(* CODESYS project 17.08.01_vi_gwp_library.library
   Title: GWP Library
   Author: ShgB
   Placeholder: GWP Library
   Version: 17.8.1
   Company: Viessmann

Project tree, tasks and I/O mapping:
  libraries: Tc2_Standard, * (Beckhoff Automation GmbH); Tc2_System, * (Beckhoff Automation GmbH); Tc2_Utilities, * (Beckhoff Automation GmbH)
  Allgemein/
    function block Alarm [ST]
    function block COUNT [ST]
    function block MUX_B [ST]
    function block MUX_D_INT [ST]
    function block MUX_D_REAL [ST]
    function block NULL [ST]
    function block SWITCH_INT [ST]
    function block SWITCH_REAL [ST]
    function block Toggle [ST]
  Converters/
    function block Converter2Punkt [ST]
    function block Int_to_Druck [ST]
    function block Int_to_Temperature [ST]
    function block Prozent_to_Int [ST]
    function block Time_to_Timestruct [ST]
    function block Timestruct_to_Time [ST]
  Druck_Temp/
    function block R1234ze [ST]
    function block R134a [ST]
    function block R410a [ST]
  Globale Variablen/
    data type AL_Eintrag
    text list Alarme
    global variables Globale_Uhr
    global variables Nassdampftabelle
    global variables SW_ALZ
    data type SW_Einsatzgrenzen
    global variables Visu
  Handschaltungen/
    function block HS_Bool [ST]
    function block HS_Int [ST]
    function block HS_Real [ST]
  Heizen_Kuehlen/
    function block FG_Heizen [ST]
    function block FG_Kuehlen [ST]
    function block GR_2 [ST]
    function block GR_4_mit_RE [ST]
    function block GR_4_ohne_RE [ST]
    function block REG2_HEIZEN [ST]
    function block REG2_KUEHLEN [ST]
    function block RT_AT_48 [ST]
  Initialisierung/
    function block Globale_Zeit [ST]
  Math/
    function block Average [ST]
    function block Filter [ST]
    function block Maximum [ST]
    function block Minimun [ST]
    function block Range [ST]
    function block Timestruct_Kleiner_Gleich_Timestruct [ST]
  Memory/
    function block Logger [ST]
  Regler/
    function block EEV [ST]
    function block PIDRegler [ST]
    function block PIRegler [ST]
    function block PRegler [ST]
  Timer/
    function block BLINK_A [ST]
    function block BLINK_S [ST]
    function block PULSE [ST]
    function block TOF_Reset [ST]
    function block TON_Reset [ST]
    function block Work [ST]
    function block XPULSE [ST]
  Uhren/
    function block ABS_Bool [ST]
    function block ABS_Int [ST]
    function block ABS_Real [ST]
    function block CLK_D [ST]
    function block CLK_I [ST]
    function block CLK_M [ST]
    function block CLK_W [ST]
    function block CLK_W7 [ST]
    function block CLK_Y [ST]
    function block FerienPRG [ST]
  Verdichter/
    function block Einsatzgrenzen [ST]
    visualisation Einsatzgrenzen
    function block FIFO [ST]
    function block SA_Scroll [ST]
  Version/
    global variables Global_Version
  text list GlobalTextList
*)

// Globale Variablen/AL_Eintrag
TYPE AL_Eintrag :
STRUCT
	x_Aktiv: BOOL;
	i_ID: INT;
	t_TimeOn: DT;
	i_TextIndex: INT;
	t_TimeOff:DT;
END_STRUCT
END_TYPE

// Globale Variablen/SW_Einsatzgrenzen
TYPE SW_Einsatzgrenzen :
STRUCT
	f_SW_EG_MinVerd:REAL;
	f_SW_EG_MaxVerd:REAL;
	f_SW_EG_MinKond:REAL;
	f_SW_EG_MaxKond:REAL;
	f_SW_EG_BVerd:REAL;
	f_SW_EG_BKond:REAL;
	f_SW_EG_CKond:REAL;
	f_SW_EG_DKond:REAL;
	f_SW_EG_EVerd:REAL;
	f_SW_EG_FVerd:REAL;
	f_SW_EG_GKond:REAL;
END_STRUCT
END_TYPE

// Globale Variablen/Globale_Uhr
{attribute 'qualified_only'}
VAR_GLOBAL
//aktuelle Uhrzeit
	   systemtimestruct	:timestruct;   
	   systemDateAndTime:dt;
END_VAR

// Globale Variablen/Nassdampftabelle
{attribute 'qualified_only'}
VAR_GLOBAL
END_VAR
VAR_GLOBAL CONSTANT
	// Arrayposition entspricht dem absoluten Druck. Z.B. 1.00bara => 0.00bar Überdruck => Arrayposition 100
	R410a: ARRAY [0..5100] OF INT := [-805,-802,-799,-796,-799,-795,-792,-789,-785,-782,-779,-776,-772,-769,-766,-762,-759,-756,-752,-749,-746,-743,-739,-736,-733,-729,-726,-723,-719,-716,-713,-710,-706,-703,-700,-703,-698,-694,-690,-685,-681,-677,-673,-669,-666,-662,-658,-654,-651,-647,-644,-641,-637,-634,-631,-628,-624,-621,-618,-615,-612,-609,-606,-604,-601,-598,-595,-592,-590,-587,-585,-582,-579,-577,-574,-572,-569,-567,-565,-562,-560,-558,-555,-553,-551,-548,-546,-544,-542,-540,-537,-535,-533,-531,-529,-527,-525,-523,-521,-519,-517,-515,-513,-511,-509,-507,-506,-504,-502,-500,-498,-496,-495,-493,-491,-489,-488,-486,-484,-482,-481,-479,-477,-476,-474,-472,-471,-469,-467,-466,-464,-463,-461,-459,-458,-456,-455,-453,-452,-450,-449,-447,-446,-444,-443,-441,-440,-438,-437,-436,-434,-433,-431,-430,-428,-427,-426,-424,-423,-422,-420,-419,-418,-416,-415,-414,-412,-411,-410,-408,-407,-406,-404,-403,-402,-401,-399,-398,-397,-396,-394,-393,-392,-391,-390,-388,-387,-386,-385,-384,-382,-381,-380,-379,-378,-377,-375,-374,-373,-372,-371,-370,-369,-367,-366,-365,-364,-363,-362,-361,-360,-359,-357,-356,-355,-354,-353,-352,-351,-350,-349,-348,-347,-346,-345,-344,-343,-342,-341,-340,-339,-338,-337,-336,-335,-334,-333,-332,-331,-330,-329,-328,-327,-326,-325,-324,-323,-322,-321,-320,-319,-318,-317,-316,-315,-314,-313,-312,-311,-310,-309,-309,-308,-307,-306,-305,-304,-303,-302,-301,-300,-299,-299,-298,-297,-296,-295,-294,-293,-292,-291,-291,-290,-289,-288,-287,-286,-285,-285,-284,-283,-282,-281,-280,-279,-279,-278,-277,-276,-275,-274,-274,-273,-272,-271,-270,-269,-269,-268,-267,-266,-265,-265,-264,-263,-262,-261,-261,-260,-259,-258,-257,-257,-256,-255,-254,-254,-253,-252,-251,-250,-250,-249,-248,-247,-247,-246,-245,-244,-244,-243,-242,-241,-241,-240,-239,-238,-238,-237,-236,-235,-235,-234,-233,-232,-232,-231,-230,-230,-229,-228,-227,-227,-226,-225,-225,-224,-223,-222,-222,-221,-220,-220,-219,-218,-218,-217,-216,-215,-215,-214,-213,-213,-212,-211,-211,-210,-209,-209,-208,-207,-207,-206,-205,-204,-204,-203,-202,-202,-201,-200,-200,-199,-199,-198,-197,-197,-196,-195,-195,-194,-193,-193,-192,-191,-191,-190,-189,-189,-188,-187,-187,-186,-186,-185,-184,-184,-183,-182,-182,-181,-180,-180,-179,-179,-178,-177,-177,-176,-176,-175,-174,-174,-173,-172,-172,-171,-171,-170,-169,-169,-168,-168,-167,-166,-166,-165,-165,-164,-163,-163,-162,-162,-161,-160,-160,-159,-159,-158,-157,-157,-156,-156,-155,-154,-154,-153,-153,-152,-152,-151,-150,-150,-149,-149,-148,-148,-147,-146,-146,-145,-145,-144,-144,-143,-142,-142,-141,-141,-140,-140,-139,-139,-138,-137,-137,-136,-136,-135,-135,-134,-134,-133,-132,-132,-131,-131,-130,-130,-129,-129,-128,-128,-127,-126,-126,-125,-125,-124,-124,-123,-123,-122,-122,-121,-121,-120,-119,-119,-118,-118,-117,-117,-116,-116,-115,-115,-114,-114,-113,-113,-112,-112,-111,-111,-110,-110,-109,-108,-108,-107,-107,-106,-106,-105,-105,-104,-104,-103,-103,-102,-102,-101,-101,-100,-100,-99,-99,-98,-98,-97,-97,-96,-96,-95,-95,-94,-94,-93,-93,-92,-92,-91,-91,-90,-90,-89,-89,-88,-88,-87,-87,-86,-86,-86,-85,-85,-84,-84,-83,-83,-82,-82,-81,-81,-80,-80,-79,-79,-78,-78,-77,-77,-76,-76,-75,-75,-75,-74,-74,-73,-73,-72,-72,-71,-71,-70,-70,-69,-69,-68,-68,-68,-67,-67,-66,-66,-65,-65,-64,-64,-63,-63,-62,-62,-62,-61,-61,-60,-60,-59,-59,-58,-58,-57,-57,-57,-56,-56,-55,-55,-54,-54,-53,-53,-53,-52,-52,-51,-51,-50,-50,-49,-49,-49,-48,-48,-47,-47,-46,-46,-45,-45,-45,-44,-44,-43,-43,-42,-42,-42,-41,-41,-40,-40,-39,-39,-39,-38,-38,-37,-37,-36,-36,-35,-35,-35,-34,-34,-33,-33,-33,-32,-32,-31,-31,-30,-30,-30,-29,-29,-28,-28,-27,-27,-27,-26,-26,-25,-25,-25,-24,-24,-23,-23,-22,-22,-22,-21,-21,-20,-20,-20,-19,-19,-18,-18,-18,-17,-17,-16,-16,-15,-15,-15,-14,-14,-13,-13,-13,-12,-12,-11,-11,-11,-10,-10,-9,-9,-9,-8,-8,-7,-7,-7,-6,-6,-5,-5,-5,-4,-4,-3,-3,-3,-2,-2,-2,-1,-1,0,0,1,1,1,2,2,3,3,3,4,4,4,5,5,6,6,6,7,7,8,8,8,9,9,9,10,10,11,11,11,12,12,13,13,13,14,14,14,15,15,16,16,16,17,17,17,18,18,19,19,19,20,20,20,21,21,22,22,22,23,23,23,24,24,25,25,25,26,26,26,27,27,27,28,28,29,29,29,30,30,30,31,31,31,32,32,33,33,33,34,34,34,35,35,35,36,36,37,37,37,38,38,38,39,39,39,40,40,40,41,41,42,42,42,43,43,43,44,44,44,45,45,45,46,46,46,47,47,48,48,48,49,49,49,50,50,50,51,51,51,52,52,52,53,53,53,54,54,54,55,55,56,56,56,57,57,57,58,58,58,59,59,59,60,60,60,61,61,61,62,62,62,63,63,63,64,64,64,65,65,65,66,66,66,67,67,67,68,68,68,69,69,69,70,70,70,71,71,71,72,72,72,73,73,73,74,74,74,75,75,75,76,76,76,77,77,77,78,78,78,79,79,79,80,80,80,81,81,81,82,82,82,83,83,83,83,84,84,84,85,85,85,86,86,86,87,87,87,88,88,88,89,89,89,90,90,90,91,91,91,91,92,92,92,93,93,93,94,94,94,95,95,95,96,96,96,97,97,97,97,98,98,98,99,99,99,100,100,100,101,101,101,101,102,102,102,103,103,103,104,104,104,105,105,105,105,106,106,106,107,107,107,108,108,108,109,109,109,109,110,110,110,111,111,111,112,112,112,113,113,113,113,114,114,114,115,115,115,116,116,116,116,117,117,117,118,118,118,119,119,119,119,120,120,120,121,121,121,121,122,122,122,123,123,123,124,124,124,124,125,125,125,126,126,126,127,127,127,127,128,128,128,129,129,129,129,130,130,130,131,131,131,131,132,132,132,133,133,133,133,134,134,134,135,135,135,136,136,136,136,137,137,137,138,138,138,138,139,139,139,140,140,140,140,141,141,141,142,142,142,142,143,143,143,143,144,144,144,145,145,145,145,146,146,146,147,147,147,147,148,148,148,149,149,149,149,150,150,150,151,151,151,151,152,152,152,152,153,153,153,154,154,154,154,155,155,155,155,156,156,156,157,157,157,157,158,158,158,159,159,159,159,160,160,160,160,161,161,161,162,162,162,162,163,163,163,163,164,164,164,164,165,165,165,166,166,166,166,167,167,167,167,168,168,168,169,169,169,169,170,170,170,170,171,171,171,171,172,172,172,173,173,173,173,174,174,174,174,175,175,175,175,176,176,176,177,177,177,177,178,178,178,178,179,179,179,179,180,180,180,180,181,181,181,181,182,182,182,183,183,183,183,184,184,184,184,185,185,185,185,186,186,186,186,187,187,187,187,188,188,188,188,189,189,189,189,190,190,190,191,191,191,191,192,192,192,192,193,193,193,193,194,194,194,194,195,195,195,195,196,196,196,196,197,197,197,197,198,198,198,198,199,199,199,199,200,200,200,200,201,201,201,201,202,202,202,202,203,203,203,203,204,204,204,204,205,205,205,205,206,206,206,206,207,207,207,207,208,208,208,208,209,209,209,209,210,210,210,210,211,211,211,211,212,212,212,212,213,213,213,213,214,214,214,214,214,215,215,215,215,216,216,216,216,217,217,217,217,218,218,218,218,219,219,219,219,220,220,220,220,221,221,221,221,221,222,222,222,222,223,223,223,223,224,224,224,224,225,225,225,225,226,226,226,226,227,227,227,227,227,228,228,228,228,229,229,229,229,230,230,230,230,231,231,231,231,231,232,232,232,232,233,233,233,233,234,234,234,234,235,235,235,235,235,236,236,236,236,237,237,237,237,238,238,238,238,238,239,239,239,239,240,240,240,240,241,241,241,241,241,242,242,242,242,243,243,243,243,244,244,244,244,244,245,245,245,245,246,246,246,246,247,247,247,247,247,248,248,248,248,249,249,249,249,249,250,250,250,250,251,251,251,251,252,252,252,252,252,253,253,253,253,254,254,254,254,254,255,255,255,255,256,256,256,256,256,257,257,257,257,258,258,258,258,258,259,259,259,259,260,260,260,260,260,261,261,261,261,262,262,262,262,262,263,263,263,263,264,264,264,264,264,265,265,265,265,266,266,266,266,266,267,267,267,267,268,268,268,268,268,269,269,269,269,270,270,270,270,270,271,271,271,271,271,272,272,272,272,273,273,273,273,273,274,274,274,274,275,275,275,275,275,276,276,276,276,276,277,277,277,277,278,278,278,278,278,279,279,279,279,279,280,280,280,280,281,281,281,281,281,282,282,282,282,282,283,283,283,283,283,284,284,284,284,285,285,285,285,285,286,286,286,286,286,287,287,287,287,288,288,288,288,288,289,289,289,289,289,290,290,290,290,290,291,291,291,291,291,292,292,292,292,293,293,293,293,293,294,294,294,294,294,295,295,295,295,295,296,296,296,296,296,297,297,297,297,298,298,298,298,298,299,299,299,299,299,300,300,300,300,300,301,301,301,301,301,302,302,302,302,302,303,303,303,303,303,304,304,304,304,304,305,305,305,305,305,306,306,306,306,307,307,307,307,307,308,308,308,308,308,309,309,309,309,309,310,310,310,310,310,311,311,311,311,311,312,312,312,312,312,313,313,313,313,313,314,314,314,314,314,315,315,315,315,315,316,316,316,316,316,317,317,317,317,317,318,318,318,318,318,319,319,319,319,319,320,320,320,320,320,321,321,321,321,321,322,322,322,322,322,322,323,323,323,323,323,324,324,324,324,324,325,325,325,325,325,326,326,326,326,326,327,327,327,327,327,328,328,328,328,328,329,329,329,329,329,330,330,330,330,330,330,331,331,331,331,331,332,332,332,332,332,333,333,333,333,333,334,334,334,334,334,335,335,335,335,335,336,336,336,336,336,336,337,337,337,337,337,338,338,338,338,338,339,339,339,339,339,340,340,340,340,340,340,341,341,341,341,341,342,342,342,342,342,343,343,343,343,343,344,344,344,344,344,344,345,345,345,345,345,346,346,346,346,346,347,347,347,347,347,347,348,348,348,348,348,349,349,349,349,349,350,350,350,350,350,350,351,351,351,351,351,352,352,352,352,352,352,353,353,353,353,353,354,354,354,354,354,355,355,355,355,355,355,356,356,356,356,356,357,357,357,357,357,357,358,358,358,358,358,359,359,359,359,359,360,360,360,360,360,360,361,361,361,361,361,362,362,362,362,362,362,363,363,363,363,363,364,364,364,364,364,364,365,365,365,365,365,366,366,366,366,366,366,367,367,367,367,367,368,368,368,368,368,368,369,369,369,369,369,370,370,370,370,370,370,371,371,371,371,371,371,372,372,372,372,372,373,373,373,373,373,373,374,374,374,374,374,375,375,375,375,375,375,376,376,376,376,376,376,377,377,377,377,377,378,378,378,378,378,378,379,379,379,379,379,379,380,380,380,380,380,381,381,381,381,381,381,382,382,382,382,382,382,383,383,383,383,383,384,384,384,384,384,384,385,385,385,385,385,385,386,386,386,386,386,387,387,387,387,387,387,388,388,388,388,388,388,389,389,389,389,389,389,390,390,390,390,390,391,391,391,391,391,391,392,392,392,392,392,392,393,393,393,393,393,393,394,394,394,394,394,394,395,395,395,395,395,395,396,396,396,396,396,397,397,397,397,397,397,398,398,398,398,398,398,399,399,399,399,399,399,400,400,400,400,400,400,401,401,401,401,401,401,402,402,402,402,402,402,403,403,403,403,403,404,404,404,404,404,404,405,405,405,405,405,405,406,406,406,406,406,406,407,407,407,407,407,407,408,408,408,408,408,408,409,409,409,409,409,409,410,410,410,410,410,410,411,411,411,411,411,411,412,412,412,412,412,412,413,413,413,413,413,413,414,414,414,414,414,414,415,415,415,415,415,415,416,416,416,416,416,416,417,417,417,417,417,417,418,418,418,418,418,418,418,419,419,419,419,419,419,420,420,420,420,420,420,421,421,421,421,421,421,422,422,422,422,422,422,423,423,423,423,423,423,424,424,424,424,424,424,425,425,425,425,425,425,426,426,426,426,426,426,426,427,427,427,427,427,427,428,428,428,428,428,428,429,429,429,429,429,429,430,430,430,430,430,430,431,431,431,431,431,431,431,432,432,432,432,432,432,433,433,433,433,433,433,434,434,434,434,434,434,435,435,435,435,435,435,435,436,436,436,436,436,436,437,437,437,437,437,437,438,438,438,438,438,438,439,439,439,439,439,439,439,440,440,440,440,440,440,441,441,441,441,441,441,442,442,442,442,442,442,442,443,443,443,443,443,443,444,444,444,444,444,444,445,445,445,445,445,445,445,446,446,446,446,446,446,447,447,447,447,447,447,447,448,448,448,448,448,448,449,449,449,449,449,449,450,450,450,450,450,450,450,451,451,451,451,451,451,452,452,452,452,452,452,452,453,453,453,453,453,453,454,454,454,454,454,454,454,455,455,455,455,455,455,456,456,456,456,456,456,456,457,457,457,457,457,457,458,458,458,458,458,458,458,459,459,459,459,459,459,460,460,460,460,460,460,460,461,461,461,461,461,461,461,462,462,462,462,462,462,463,463,463,463,463,463,463,464,464,464,464,464,464,465,465,465,465,465,465,465,466,466,466,466,466,466,466,467,467,467,467,467,467,468,468,468,468,468,468,468,469,469,469,469,469,469,469,470,470,470,470,470,470,471,471,471,471,471,471,471,472,472,472,472,472,472,472,473,473,473,473,473,473,474,474,474,474,474,474,474,475,475,475,475,475,475,475,476,476,476,476,476,476,476,477,477,477,477,477,477,478,478,478,478,478,478,478,479,479,479,479,479,479,479,480,480,480,480,480,480,480,481,481,481,481,481,481,482,482,482,482,482,482,482,483,483,483,483,483,483,483,484,484,484,484,484,484,484,485,485,485,485,485,485,485,486,486,486,486,486,486,486,487,487,487,487,487,487,487,488,488,488,488,488,488,488,489,489,489,489,489,489,490,490,490,490,490,490,490,491,491,491,491,491,491,491,492,492,492,492,492,492,492,493,493,493,493,493,493,493,494,494,494,494,494,494,494,495,495,495,495,495,495,495,496,496,496,496,496,496,496,497,497,497,497,497,497,497,498,498,498,498,498,498,498,499,499,499,499,499,499,499,500,500,500,500,500,500,500,501,501,501,501,501,501,501,502,502,502,502,502,502,502,503,503,503,503,503,503,503,504,504,504,504,504,504,504,504,505,505,505,505,505,505,505,506,506,506,506,506,506,506,507,507,507,507,507,507,507,508,508,508,508,508,508,508,509,509,509,509,509,509,509,510,510,510,510,510,510,510,511,511,511,511,511,511,511,511,512,512,512,512,512,512,512,513,513,513,513,513,513,513,514,514,514,514,514,514,514,515,515,515,515,515,515,515,516,516,516,516,516,516,516,516,517,517,517,517,517,517,517,518,518,518,518,518,518,518,519,519,519,519,519,519,519,519,520,520,520,520,520,520,520,521,521,521,521,521,521,521,522,522,522,522,522,522,522,523,523,523,523,523,523,523,523,524,524,524,524,524,524,524,525,525,525,525,525,525,525,525,526,526,526,526,526,526,526,527,527,527,527,527,527,527,528,528,528,528,528,528,528,528,529,529,529,529,529,529,529,530,530,530,530,530,530,530,530,531,531,531,531,531,531,531,532,532,532,532,532,532,532,533,533,533,533,533,533,533,533,534,534,534,534,534,534,534,535,535,535,535,535,535,535,535,536,536,536,536,536,536,536,537,537,537,537,537,537,537,537,538,538,538,538,538,538,538,538,539,539,539,539,539,539,539,540,540,540,540,540,540,540,540,541,541,541,541,541,541,541,542,542,542,542,542,542,542,542,543,543,543,543,543,543,543,544,544,544,544,544,544,544,544,545,545,545,545,545,545,545,545,546,546,546,546,546,546,546,547,547,547,547,547,547,547,547,548,548,548,548,548,548,548,548,549,549,549,549,549,549,549,550,550,550,550,550,550,550,550,551,551,551,551,551,551,551,551,552,552,552,552,552,552,552,553,553,553,553,553,553,553,553,554,554,554,554,554,554,554,554,555,555,555,555,555,555,555,555,556,556,556,556,556,556,556,556,557,557,557,557,557,557,557,558,558,558,558,558,558,558,558,559,559,559,559,559,559,559,559,560,560,560,560,560,560,560,560,561,561,561,561,561,561,561,561,562,562,562,562,562,562,562,562,563,563,563,563,563,563,563,564,564,564,564,564,564,564,564,565,565,565,565,565,565,565,565,566,566,566,566,566,566,566,566,567,567,567,567,567,567,567,567,568,568,568,568,568,568,568,568,569,569,569,569,569,569,569,569,570,570,570,570,570,570,570,570,571,571,571,571,571,571,571,571,572,572,572,572,572,572,572,572,573,573,573,573,573,573,573,573,574,574,574,574,574,574,574,574,575,575,575,575,575,575,575,575,576,576,576,576,576,576,576,576,577,577,577,577,577,577,577,577,578,578,578,578,578,578,578,578,579,579,579,579,579,579,579,579,580,580,580,580,580,580,580,580,580,581,581,581,581,581,581,581,581,582,582,582,582,582,582,582,582,583,583,583,583,583,583,583,583,584,584,584,584,584,584,584,584,585,585,585,585,585,585,585,585,586,586,586,586,586,586,586,586,586,587,587,587,587,587,587,587,587,588,588,588,588,588,588,588,588,589,589,589,589,589,589,589,589,590,590,590,590,590,590,590,590,590,591,591,591,591,591,591,591,591,592,592,592,592,592,592,592,592,593,593,593,593,593,593,593,593,593,594,594,594,594,594,594,594,594,595,595,595,595,595,595,595,595,596,596,596,596,596,596,596,596,596,597,597,597,597,597,597,597,597,598,598,598,598,598,598,598,598,599,599,599,599,599,599,599,599,599,600,600,600,600,600,600,600,600,601,601,601,601,601,601,601,601,601,602,602,602,602,602,602,602,602,603,603,603,603,603,603,603,603,604,604,604,604,604,604,604,604,604,605,605,605,605,605,605,605,605,606,606,606,606,606,606,606,606,606,607,607,607,607,607,607,607,607,608,608,608,608,608,608,608,608,608,609,609,609,609,609,609,609,609,609,610,610,610,610,610,610,610,610,611,611,611,611,611,611,611,611,611,612,612,612,612,612,612,612,612,613,613,613,613,613,613,613,613,613,614,614,614,614,614,614,614,614,614,615,615,615,615,615,615,615,615,616,616,616,616,616,616,616,616,616,617,617,617,617,617,617,617,617,617,618,618,618,618,618,618,618,618,619,619,619,619,619,619,619,619,619,620,620,620,620,620,620,620,620,620,621,621,621,621,621,621,621,621,622,622,622,622,622,622,622,622,622,623,623,623,623,623,623,623,623,623,624,624,624,624,624,624,624,624,624,625,625,625,625,625,625,625,625,625,626,626,626,626,626,626,626,626,627,627,627,627,627,627,627,627,627,628,628,628,628,628,628,628,628,628,629,629,629,629,629,629,629,629,629,630,630,630,630,630,630,630,630,630,631,631,631,631,631,631,631,631,631,632,632,632,632,632,632,632,632,632,633,633,633,633,633,633,633,633,633,634,634,634,634,634,634,634,634,634,635,635,635,635,635,635,635,635,635,636,636,636,636,636,636,636,636,636,637,637,637,637,637,637,637,637,637,638,638,638,638,638,638,638,638,638,639,639,639,639,639,639,639,639,639,640,640,640,640,640,640,640,640,640,641,641,641,641,641,641,641,641,641,642,642,642,642,642,642,642,642,642,643,643,643,643,643,643,643,643,643,644,644,644,644,644,644,644,644,644,645,645,645,645,645,645,645,645,645,646,646,646,646,646,646,646,646,646,647,647,647,647,647,647,647,647,647,648,648,648,648,648,648,648,648,648,648,649,649,649,649,649,649,649,649,649,650,650,650,650,650,650,650,650,650,651,651,651,651,651,651,651,651,651,652,652,652,652,652,652,652,652,652,652,653,653,653,653,653,653,653,653,653,654,654,654,654,654,654,654,654,654,655,655,655,655,655,655,655,655,655,656,656,656,656,656,656,656,656,656,656,657,657,657,657,657,657,657,657,657,658,658,658,658,658,658,658,658,658,659,659,659,659,659,659,659,659,659,659,660,660,660,660,660,660,660,660,660,661,661,661,661,661,661,661,661,661,661,662,662,662,662,662,662,662,662,662,663,663,663,663,663,663,663,663,663,664,664,664,664,664,664,664,664,664,664,665,665,665,665,665,665,665,665,665,666,666,666,666,666,666,666,666,666,666,667,667,667,667,667,667,667,667,667,668,668,668,668,668,668,668,668,668,668,669,669,669,669,669,669,669,669,669,670,670,670,670,670,670,670,670,670,670,671,671,671,671,671,671,671,671,671,671,672,672,672,672,672,672,672,672,672,673,673,673,673,673,673,673,673,673,673,674,674,674,674,674,674,674,674,674,675,675,675,675,675,675,675,675,675,675,676,676,676,676,676,676,676,676,676,676,677,677,677,677,677,677,677,677,677,678,678,678,678,678,678,678,678,678,678,679,679,679,679,679,679,679,679,679,679,680,680,680,680,680,680,680,680,680,680,681,681,681,681,681,681,681,681,681,682,682,682,682,682,682,682,682,682,682,683,683,683,683,683,683,683,683,683,683,684,684,684,684,684,684,684,684,684,684,685,685,685,685,685,685,685,685,685,685,686,686,686,686,686,686,686,686,686,686,687,687,687,687,687,687,687,687,687,688,688,688,688,688,688,688,688,688,688,689,689,689,689,689,689,689,689,689,689,690,690,690,690,690,690,690,690,690,690,691,691,691,691,691,691,691,691,691,691,692,692,692,692,692,692,692,692,692,692,693,693,693,693,693,693,693,693,693,693,694,694,694,694,694,694,694,694,694,694,695,695,695,695,695,695,695,695,695,695,696,696,696,696,696,696,696,696,696,696,697,697,697,697,697,697,697,697,697,697,698,698,698,698,698,698,698,698,698,698,699,699,699,699,699,699,699,699,699,699,700,700,700,700,700,700,700,700,700,700,701,701,701,701,701,701,701,701,701,701,702,702,702,702,702,702,702,702,702,702,703,703,703,703,703,703,703,703,703,703,704,704,704,704,704,704,704,704,704,704,705,705,705,705,705,705,705,705,705,705,706,706,706,706,706,706,706,706,706,706,707,707,707,707,707,707,707,707,707,707,708,708,708,708,708,708,708,708,708,708,709,709,709,709,709,709,709,709,709,709,710,710,710,710,710,710,710,710,710,710,711,711,711,711,711,711,711,711,711,711,712,712,712,712,712,712,712,712,712,712,713,713,713,713,713,713,713,713,713,713,714];
	// Arrayposition entspricht dem absoluten Druck. Z.B. 1.00bara => 0.00bar Überdruck => Arrayposition 100
	R1234ze: ARRAY [0..5100] OF INT := [-483,-481,-478,-475,-472,-470,-467,-464,-461,-459,-456,-453,-450,-448,-445,-442,-439,-437,-434,-431,-428,-426,-423,-420,-477,-470,-463,-456,-450,-443,-437,-431,-426,-420,-414,-409,-404,-399,-394,-389,-384,-379,-375,-370,-366,-361,-357,-353,-349,-345,-341,-337,-333,-329,-325,-322,-318,-314,-311,-307,-304,-300,-297,-294,-290,-287,-284,-281,-278,-275,-272,-268,-266,-263,-260,-257,-254,-251,-248,-245,-243,-240,-237,-235,-232,-229,-227,-224,-222,-219,-217,-214,-212,-209,-207,-204,-202,-200,-197,-195,-193,-191,-188,-186,-184,-182,-179,-177,-175,-173,-171,-169,-167,-164,-162,-160,-158,-156,-154,-152,-150,-148,-146,-144,-142,-140,-139,-137,-135,-133,-131,-129,-127,-125,-124,-122,-120,-118,-116,-115,-113,-111,-109,-108,-106,-104,-102,-101,-99,-97,-96,-94,-92,-91,-89,-88,-86,-84,-83,-81,-79,-78,-76,-75,-73,-72,-70,-69,-67,-66,-64,-62,-61,-59,-58,-57,-55,-54,-52,-51,-49,-48,-46,-45,-43,-42,-41,-39,-38,-36,-35,-34,-32,-31,-30,-28,-27,-25,-24,-23,-21,-20,-19,-17,-16,-15,-14,-12,-11,-10,-8,-7,-6,-5,-3,-2,-1,1,2,3,4,6,7,8,9,10,12,13,14,15,17,18,19,20,21,22,24,25,26,27,28,29,31,32,33,34,35,36,37,39,40,41,42,43,44,45,46,47,49,50,51,52,53,54,55,56,57,58,59,60,62,63,64,65,66,67,68,69,70,71,72,73,74,75,76,77,78,79,80,81,82,83,84,85,86,87,88,89,90,91,92,93,94,95,96,97,98,99,100,101,102,103,104,104,105,106,107,108,109,110,111,112,113,114,115,116,117,117,118,119,120,121,122,123,124,125,126,127,127,128,129,130,131,132,133,134,134,135,136,137,138,139,140,141,141,142,143,144,145,146,147,147,148,149,150,151,152,152,153,154,155,156,157,157,158,159,160,161,162,162,163,164,165,166,166,167,168,169,170,170,171,172,173,174,174,175,176,177,178,178,179,180,181,181,182,183,184,185,185,186,187,188,188,189,190,191,192,192,193,194,195,195,196,197,198,198,199,200,201,201,202,203,204,204,205,206,206,207,208,209,209,210,211,212,212,213,214,214,215,216,217,217,218,219,219,220,221,222,222,223,224,224,225,226,227,227,228,229,229,230,231,231,232,233,233,234,235,236,236,237,238,238,239,240,240,241,242,242,243,244,244,245,246,246,247,248,248,249,250,250,251,252,252,253,254,254,255,256,256,257,258,258,259,260,260,261,261,262,263,263,264,265,265,266,267,267,268,269,269,270,270,271,272,272,273,274,274,275,275,276,277,277,278,279,279,280,280,281,282,282,283,284,284,285,285,286,287,287,288,288,289,290,290,291,291,292,293,293,294,294,295,296,296,297,297,298,299,299,300,300,301,302,302,303,303,304,305,305,306,306,307,308,308,309,309,310,310,311,312,312,313,313,314,314,315,316,316,317,317,318,318,319,320,320,321,321,322,322,323,324,324,325,325,326,326,327,327,328,329,329,330,330,331,331,332,332,333,334,334,335,335,336,336,337,337,338,339,339,340,340,341,341,342,342,343,343,344,344,345,346,346,347,347,348,348,349,349,350,350,351,351,352,352,353,354,354,355,355,356,356,357,357,358,358,359,359,360,360,361,361,362,362,363,363,364,365,365,366,366,367,367,368,368,369,369,370,370,371,371,372,372,373,373,374,374,375,375,376,376,377,377,378,378,379,379,380,380,381,381,382,382,383,383,384,384,385,385,386,386,387,387,388,388,389,389,390,390,391,391,392,392,393,393,394,394,395,395,395,396,396,397,397,398,398,399,399,400,400,401,401,402,402,403,403,404,404,405,405,406,406,407,407,407,408,408,409,409,410,410,411,411,412,412,413,413,414,414,414,415,415,416,416,417,417,418,418,419,419,420,420,421,421,421,422,422,423,423,424,424,425,425,426,426,426,427,427,428,428,429,429,430,430,431,431,431,432,432,433,433,434,434,435,435,435,436,436,437,437,438,438,439,439,439,440,440,441,441,442,442,443,443,443,444,444,445,445,446,446,447,447,447,448,448,449,449,450,450,450,451,451,452,452,453,453,453,454,454,455,455,456,456,456,457,457,458,458,459,459,459,460,460,461,461,462,462,462,463,463,464,464,465,465,465,466,466,467,467,467,468,468,469,469,470,470,470,471,471,472,472,472,473,473,474,474,475,475,475,476,476,477,477,477,478,478,479,479,479,480,480,481,481,482,482,482,483,483,484,484,484,485,485,486,486,486,487,487,488,488,488,489,489,490,490,490,491,491,492,492,492,493,493,494,494,494,495,495,496,496,496,497,497,498,498,498,499,499,500,500,500,501,501,502,502,502,503,503,503,504,504,505,505,505,506,506,507,507,507,508,508,509,509,509,510,510,510,511,511,512,512,512,513,513,514,514,514,515,515,515,516,516,517,517,517,518,518,519,519,519,520,520,520,521,521,522,522,522,523,523,523,524,524,525,525,525,526,526,526,527,527,528,528,528,529,529,529,530,530,531,531,531,532,532,532,533,533,534,534,534,535,535,535,536,536,536,537,537,538,538,538,539,539,539,540,540,540,541,541,542,542,542,543,543,543,544,544,544,545,545,546,546,546,547,547,547,548,548,548,549,549,550,550,550,551,551,551,552,552,552,553,553,553,554,554,555,555,555,556,556,556,557,557,557,558,558,558,559,559,559,560,560,561,561,561,562,562,562,563,563,563,564,564,564,565,565,565,566,566,566,567,567,568,568,568,569,569,569,570,570,570,571,571,571,572,572,572,573,573,573,574,574,574,575,575,575,576,576,576,577,577,577,578,578,579,579,579,580,580,580,581,581,581,582,582,582,583,583,583,584,584,584,585,585,585,586,586,586,587,587,587,588,588,588,589,589,589,590,590,590,591,591,591,592,592,592,593,593,593,594,594,594,595,595,595,596,596,596,597,597,597,598,598,598,599,599,599,600,600,600,601,601,601,601,602,602,602,603,603,603,604,604,604,605,605,605,606,606,606,607,607,607,608,608,608,609,609,609,610,610,610,611,611,611,612,612,612,612,613,613,613,614,614,614,615,615,615,616,616,616,617,617,617,618,618,618,619,619,619,619,620,620,620,621,621,621,622,622,622,623,623,623,624,624,624,625,625,625,625,626,626,626,627,627,627,628,628,628,629,629,629,629,630,630,630,631,631,631,632,632,632,633,633,633,634,634,634,634,635,635,635,636,636,636,637,637,637,638,638,638,638,639,639,639,640,640,640,641,641,641,641,642,642,642,643,643,643,644,644,644,644,645,645,645,646,646,646,647,647,647,648,648,648,648,649,649,649,650,650,650,651,651,651,651,652,652,652,653,653,653,653,654,654,654,655,655,655,656,656,656,656,657,657,657,658,658,658,659,659,659,659,660,660,660,661,661,661,661,662,662,662,663,663,663,664,664,664,664,665,665,665,666,666,666,666,667,667,667,668,668,668,668,669,669,669,670,670,670,670,671,671,671,672,672,672,673,673,673,673,674,674,674,675,675,675,675,676,676,676,677,677,677,677,678,678,678,679,679,679,679,680,680,680,681,681,681,681,682,682,682,683,683,683,683,684,684,684,684,685,685,685,686,686,686,686,687,687,687,688,688,688,688,689,689,689,690,690,690,690,691,691,691,691,692,692,692,693,693,693,693,694,694,694,695,695,695,695,696,696,696,696,697,697,697,698,698,698,698,699,699,699,700,700,700,700,701,701,701,701,702,702,702,703,703,703,703,704,704,704,704,705,705,705,706,706,706,706,707,707,707,707,708,708,708,709,709,709,709,710,710,710,710,711,711,711,711,712,712,712,713,713,713,713,714,714,714,714,715,715,715,716,716,716,716,717,717,717,717,718,718,718,718,719,719,719,719,720,720,720,721,721,721,721,722,722,722,722,723,723,723,723,724,724,724,725,725,725,725,726,726,726,726,727,727,727,727,728,728,728,728,729,729,729,730,730,730,730,731,731,731,731,732,732,732,732,733,733,733,733,734,734,734,734,735,735,735,735,736,736,736,737,737,737,737,738,738,738,738,739,739,739,739,740,740,740,740,741,741,741,741,742,742,742,742,743,743,743,743,744,744,744,744,745,745,745,745,746,746,746,746,747,747,747,748,748,748,748,749,749,749,749,750,750,750,750,751,751,751,751,752,752,752,752,753,753,753,753,754,754,754,754,755,755,755,755,756,756,756,756,757,757,757,757,758,758,758,758,759,759,759,759,760,760,760,760,761,761,761,761,762,762,762,762,763,763,763,763,764,764,764,764,764,765,765,765,765,766,766,766,766,767,767,767,767,768,768,768,768,769,769,769,769,770,770,770,770,771,771,771,771,772,772,772,772,773,773,773,773,774,774,774,774,775,775,775,775,775,776,776,776,776,777,777,777,777,778,778,778,778,779,779,779,779,780,780,780,780,781,781,781,781,781,782,782,782,782,783,783,783,783,784,784,784,784,785,785,785,785,786,786,786,786,786,787,787,787,787,788,788,788,788,789,789,789,789,790,790,790,790,791,791,791,791,791,792,792,792,792,793,793,793,793,794,794,794,794,795,795,795,795,795,796,796,796,796,797,797,797,797,798,798,798,798,798,799,799,799,799,800,800,800,800,801,801,801,801,802,802,802,802,802,803,803,803,803,804,804,804,804,805,805,805,805,805,806,806,806,806,807,807,807,807,807,808,808,808,808,809,809,809,809,810,810,810,810,810,811,811,811,811,812,812,812,812,813,813,813,813,813,814,814,814,814,815,815,815,815,815,816,816,816,816,817,817,817,817,818,818,818,818,818,819,819,819,819,820,820,820,820,820,821,821,821,821,822,822,822,822,822,823,823,823,823,824,824,824,824,824,825,825,825,825,826,826,826,826,826,827,827,827,827,828,828,828,828,828,829,829,829,829,830,830,830,830,830,831,831,831,831,832,832,832,832,832,833,833,833,833,834,834,834,834,834,835,835,835,835,836,836,836,836,836,837,837,837,837,837,838,838,838,838,839,839,839,839,839,840,840,840,840,841,841,841,841,841,842,842,842,842,842,843,843,843,843,844,844,844,844,844,845,845,845,845,846,846,846,846,846,847,847,847,847,847,848,848,848,848,849,849,849,849,849,850,850,850,850,850,851,851,851,851,852,852,852,852,852,853,853,853,853,853,854,854,854,854,855,855,855,855,855,856,856,856,856,856,857,857,857,857,857,858,858,858,858,859,859,859,859,859,860,860,860,860,860,861,861,861,861,861,862,862,862,862,863,863,863,863,863,864,864,864,864,864,865,865,865,865,865,866,866,866,866,866,867,867,867,867,868,868,868,868,868,869,869,869,869,869,870,870,870,870,870,871,871,871,871,871,872,872,872,872,873,873,873,873,873,874,874,874,874,874,875,875,875,875,875,876,876,876,876,876,877,877,877,877,877,878,878,878,878,878,879,879,879,879,879,880,880,880,880,880,881,881,881,881,882,882,882,882,882,883,883,883,883,883,884,884,884,884,884,885,885,885,885,885,886,886,886,886,886,887,887,887,887,887,888,888,888,888,888,889,889,889,889,889,890,890,890,890,890,891,891,891,891,891,892,892,892,892,892,893,893,893,893,893,894,894,894,894,894,895,895,895,895,895,896,896,896,896,896,897,897,897,897,897,898,898,898,898,898,899,899,899,899,899,900,900,900,900,900,901,901,901,901,901,902,902,902,902,902,903,903,903,903,903,903,904,904,904,904,904,905,905,905,905,905,906,906,906,906,906,907,907,907,907,907,908,908,908,908,908,909,909,909,909,909,910,910,910,910,910,911,911,911,911,911,911,912,912,912,912,912,913,913,913,913,913,914,914,914,914,914,915,915,915,915,915,916,916,916,916,916,916,917,917,917,917,917,918,918,918,918,918,919,919,919,919,919,920,920,920,920,920,921,921,921,921,921,921,922,922,922,922,922,923,923,923,923,923,924,924,924,924,924,925,925,925,925,925,925,926,926,926,926,926,927,927,927,927,927,928,928,928,928,928,928,929,929,929,929,929,930,930,930,930,930,931,931,931,931,931,931,932,932,932,932,932,933,933,933,933,933,934,934,934,934,934,934,935,935,935,935,935,936,936,936,936,936,937,937,937,937,937,937,938,938,938,938,938,939,939,939,939,939,939,940,940,940,940,940,941,941,941,941,941,942,942,942,942,942,942,943,943,943,943,943,944,944,944,944,944,944,945,945,945,945,945,946,946,946,946,946,946,947,947,947,947,947,948,948,948,948,948,949,949,949,949,949,949,950,950,950,950,950,951,951,951,951,951,951,952,952,952,952,952,953,953,953,953,953,953,954,954,954,954,954,954,955,955,955,955,955,956,956,956,956,956,956,957,957,957,957,957,958,958,958,958,958,958,959,959,959,959,959,960,960,960,960,960,960,961,961,961,961,961,961,962,962,962,962,962,963,963,963,963,963,963,964,964,964,964,964,965,965,965,965,965,965,966,966,966,966,966,966,967,967,967,967,967,968,968,968,968,968,968,969,969,969,969,969,969,970,970,970,970,970,971,971,971,971,971,971,972,972,972,972,972,972,973,973,973,973,973,974,974,974,974,974,974,975,975,975,975,975,975,976,976,976,976,976,976,977,977,977,977,977,978,978,978,978,978,978,979,979,979,979,979,979,980,980,980,980,980,980,981,981,981,981,981,982,982,982,982,982,982,983,983,983,983,983,983,984,984,984,984,984,984,985,985,985,985,985,985,986,986,986,986,986,987,987,987,987,987,987,988,988,988,988,988,988,989,989,989,989,989,989,990,990,990,990,990,990,991,991,991,991,991,991,992,992,992,992,992,992,993,993,993,993,993,993,994,994,994,994,994,994,995,995,995,995,995,996,996,996,996,996,996,997,997,997,997,997,997,998,998,998,998,998,998,999,999,999,999,999,999,1000,1000,1000,1000,1000,1000,1001,1001,1001,1001,1001,1001,1002,1002,1002,1002,1002,1002,1003,1003,1003,1003,1003,1003,1004,1004,1004,1004,1004,1004,1005,1005,1005,1005,1005,1005,1006,1006,1006,1006,1006,1006,1007,1007,1007,1007,1007,1007,1008,1008,1008,1008,1008,1008,1009,1009,1009,1009,1009,1009,1010,1010,1010,1010,1010,1010,1011,1011,1011,1011,1011,1011,1011,1012,1012,1012,1012,1012,1012,1013,1013,1013,1013,1013,1013,1014,1014,1014,1014,1014,1014,1015,1015,1015,1015,1015,1015,1016,1016,1016,1016,1016,1016,1017,1017,1017,1017,1017,1017,1018,1018,1018,1018,1018,1018,1019,1019,1019,1019,1019,1019,1019,1020,1020,1020,1020,1020,1020,1021,1021,1021,1021,1021,1021,1022,1022,1022,1022,1022,1022,1023,1023,1023,1023,1023,1023,1024,1024,1024,1024,1024,1024,1024,1025,1025,1025,1025,1025,1025,1026,1026,1026,1026,1026,1026,1027,1027,1027,1027,1027,1027,1028,1028,1028,1028,1028,1028,1028,1029,1029,1029,1029,1029,1029,1030,1030,1030,1030,1030,1030,1031,1031,1031,1031,1031,1031,1032,1032,1032,1032,1032,1032,1032,1033,1033,1033,1033,1033,1033,1034,1034,1034,1034,1034,1034,1035,1035,1035,1035,1035,1035,1035,1036,1036,1036,1036,1036,1036,1037,1037,1037,1037,1037,1037,1038,1038,1038,1038,1038,1038,1038,1039,1039,1039,1039,1039,1039,1040,1040,1040,1040,1040,1040,1040,1041,1041,1041,1041,1041,1041,1042,1042,1042,1042,1042,1042,1043,1043,1043,1043,1043,1043,1043,1044,1044,1044,1044,1044,1044,1045,1045,1045,1045,1045,1045,1045,1046,1046,1046,1046,1046,1046,1047,1047,1047,1047,1047,1047,1047,1048,1048,1048,1048,1048,1048,1049,1049,1049,1049,1049,1049,1049,1050,1050,1050,1050,1050,1050,1051,1051,1051,1051,1051,1051,1051,1052,1052,1052,1052,1052,1052,1053,1053,1053,1053,1053,1053,1053,1054,1054,1054,1054,1054,1054,1055,1055,1055,1055,1055,1055,1055,1056,1056,1056,1056,1056,1056,1056,1057,1057,1057,1057,1057,1057,1058,1058,1058,1058,1058,1058,1058,1059,1059,1059,1059,1059,1059,1060,1060,1060,1060,1060,1060,1060,1061,1061,1061,1061,1061,1061,1061,1062,1062,1062,1062,1062,1062,1063,1063,1063,1063,1063,1063,1063,1064,1064,1064,1064,1064,1064,1064,1065,1065,1065,1065,1065,1065,1066,1066,1066,1066,1066,1066,1066,1067,1067,1067,1067,1067,1067,1067,1068,1068,1068,1068,1068,1068,1068,1069,1069,1069,1069,1069,1069,1070,1070,1070,1070,1070,1070,1070,1071,1071,1071,1071,1071,1071,1071,1072,1072,1072,1072,1072,1072,1072,1073,1073,1073,1073,1073,1073,1073,1074,1074,1074,1074,1074,1074,1075,1075,1075,1075,1075,1075,1075,1076,1076,1076,1076,1076,1076,1076,1077,1077,1077,1077,1077,1077,1077,1078,1078,1078,1078,1078,1078,1078,1079,1079,1079,1079,1079,1079,1079,1080,1080,1080,1080,1080,1080,1080,1081,1081,1081,1081,1081,1081,1081,1082,1082,1082,1082,1082,1082,1083,1083,1083,1083,1083,1083,1083,1084,1084,1084,1084,1084,1084,1084,1085,1085,1085,1085,1085,1085,1085,1086,1086,1086,1086,1086,1086,1086,1087,1087,1087,1087,1087,1087,1087,1088,1088,1088,1088,1088,1088,1088,1088,1089,1089,1089,1089,1089,1089,1089,1090,1090,1090,1090,1090,1090,1090,1091,1091,1091,1091,1091,1091,1091,1092,1092,1092,1092,1092,1092,1092,1093,1093,1093,1093];
	// Arrayposition entspricht dem absoluten Druck. Z.B. 1.00bara => 0.00bar Überdruck => Arrayposition 100
	R134a: ARRAY [0..5100] OF INT := [-571,-568,-564,-561,-558,-554,-551,-548,-544,-541,-538,-534,-531,-528,-524,-521,-517,-514,-511,-507,-504,-501,-497,-494,-491,-487,-484,-481,-477,-474,-471,-467,-464,-460,-457,-454,-450,-447,-444,-440,-437,-434,-430,-427,-424,-420,-417,-413,-410,-407,-405,-401,-397,-393,-390,-386,-383,-379,-376,-373,-369,-366,-363,-360,-357,-354,-350,-347,-344,-342,-339,-336,-333,-330,-327,-325,-322,-319,-316,-314,-311,-309,-306,-304,-301,-299,-296,-294,-291,-289,-286,-284,-282,-279,-277,-275,-273,-270,-268,-266,-264,-261,-259,-257,-255,-253,-251,-249,-247,-245,-243,-241,-239,-237,-235,-233,-231,-229,-227,-225,-223,-221,-219,-218,-216,-214,-212,-210,-208,-207,-205,-203,-201,-200,-198,-196,-194,-193,-191,-189,-188,-186,-184,-183,-181,-179,-178,-176,-175,-173,-171,-170,-168,-167,-165,-164,-162,-160,-159,-157,-156,-154,-153,-151,-150,-148,-147,-146,-144,-143,-141,-140,-138,-137,-136,-134,-133,-131,-130,-129,-127,-126,-124,-123,-122,-120,-119,-118,-116,-115,-114,-112,-111,-110,-108,-107,-106,-105,-103,-102,-101,-100,-98,-97,-96,-95,-93,-92,-91,-90,-88,-87,-86,-85,-84,-82,-81,-80,-79,-78,-76,-75,-74,-73,-72,-71,-69,-68,-67,-66,-65,-64,-63,-61,-60,-59,-58,-57,-56,-55,-54,-53,-52,-50,-49,-48,-47,-46,-45,-44,-43,-42,-41,-40,-39,-38,-37,-36,-34,-33,-32,-31,-30,-29,-28,-27,-26,-25,-24,-23,-22,-21,-20,-19,-18,-17,-16,-15,-14,-13,-12,-11,-10,-9,-8,-7,-7,-6,-5,-4,-3,-2,-1,0,1,2,3,4,5,6,7,8,9,10,10,11,12,13,14,15,16,17,18,19,19,20,21,22,23,24,25,26,27,27,28,29,30,31,32,33,34,34,35,36,37,38,39,39,40,41,42,43,44,45,45,46,47,48,49,50,50,51,52,53,54,54,55,56,57,58,58,59,60,61,62,62,63,64,65,66,66,67,68,69,70,70,71,72,73,73,74,75,76,77,77,78,79,80,80,81,82,83,83,84,85,86,86,87,88,89,89,90,91,92,92,93,94,95,95,96,97,97,98,99,100,100,101,102,102,103,104,105,105,106,107,107,108,109,110,110,111,112,112,113,114,115,115,116,117,117,118,119,119,120,121,121,122,123,123,124,125,125,126,127,128,128,129,130,130,131,132,132,133,134,134,135,136,136,137,138,138,139,139,140,141,141,142,143,143,144,145,145,146,147,147,148,149,149,150,150,151,152,152,153,154,154,155,156,156,157,157,158,159,159,160,161,161,162,162,163,164,164,165,165,166,167,167,168,169,169,170,170,171,172,172,173,173,174,175,175,176,176,177,178,178,179,179,180,181,181,182,182,183,183,184,185,185,186,186,187,188,188,189,189,190,190,191,192,192,193,193,194,195,195,196,196,197,197,198,199,199,200,200,201,201,202,202,203,204,204,205,205,206,206,207,208,208,209,209,210,210,211,211,212,212,213,214,214,215,215,216,216,217,217,218,218,219,220,220,221,221,222,222,223,223,224,224,225,225,226,227,227,228,228,229,229,230,230,231,231,232,232,233,233,234,234,235,235,236,237,237,238,238,239,239,240,240,241,241,242,242,243,243,244,244,245,245,246,246,247,247,248,248,249,249,250,250,251,251,252,252,253,253,254,254,255,255,256,256,257,257,258,258,259,259,260,260,261,261,262,262,263,263,264,264,265,265,266,266,267,267,268,268,269,269,270,270,271,271,272,272,272,273,273,274,274,275,275,276,276,277,277,278,278,279,279,280,280,281,281,282,282,282,283,283,284,284,285,285,286,286,287,287,288,288,289,289,289,290,290,291,291,292,292,293,293,294,294,295,295,295,296,296,297,297,298,298,299,299,300,300,300,301,301,302,302,303,303,304,304,304,305,305,306,306,307,307,308,308,308,309,309,310,310,311,311,312,312,312,313,313,314,314,315,315,316,316,316,317,317,318,318,319,319,319,320,320,321,321,322,322,322,323,323,324,324,325,325,325,326,326,327,327,328,328,328,329,329,330,330,331,331,331,332,332,333,333,334,334,334,335,335,336,336,336,337,337,338,338,339,339,339,340,340,341,341,341,342,342,343,343,344,344,344,345,345,346,346,346,347,347,348,348,348,349,349,350,350,350,351,351,352,352,352,353,353,354,354,355,355,355,356,356,357,357,357,358,358,359,359,359,360,360,361,361,361,362,362,362,363,363,364,364,364,365,365,366,366,366,367,367,368,368,368,369,369,370,370,370,371,371,372,372,372,373,373,373,374,374,375,375,375,376,376,377,377,377,378,378,378,379,379,380,380,380,381,381,382,382,382,383,383,383,384,384,385,385,385,386,386,386,387,387,388,388,388,389,389,389,390,390,391,391,391,392,392,392,393,393,394,394,394,395,395,395,396,396,397,397,397,398,398,398,399,399,399,400,400,401,401,401,402,402,402,403,403,403,404,404,405,405,405,406,406,406,407,407,407,408,408,409,409,409,410,410,410,411,411,411,412,412,413,413,413,414,414,414,415,415,415,416,416,416,417,417,417,418,418,419,419,419,420,420,420,421,421,421,422,422,422,423,423,423,424,424,425,425,425,426,426,426,427,427,427,428,428,428,429,429,429,430,430,430,431,431,431,432,432,433,433,433,434,434,434,435,435,435,436,436,436,437,437,437,438,438,438,439,439,439,440,440,440,441,441,441,442,442,442,443,443,443,444,444,444,445,445,445,446,446,446,447,447,447,448,448,448,449,449,449,450,450,450,451,451,451,452,452,452,453,453,453,454,454,454,455,455,455,456,456,456,457,457,457,458,458,458,459,459,459,460,460,460,461,461,461,462,462,462,463,463,463,464,464,464,464,465,465,465,466,466,466,467,467,467,468,468,468,469,469,469,470,470,470,471,471,471,472,472,472,473,473,473,473,474,474,474,475,475,475,476,476,476,477,477,477,478,478,478,479,479,479,479,480,480,480,481,481,481,482,482,482,483,483,483,484,484,484,484,485,485,485,486,486,486,487,487,487,488,488,488,488,489,489,489,490,490,490,491,491,491,492,492,492,492,493,493,493,494,494,494,495,495,495,496,496,496,496,497,497,497,498,498,498,499,499,499,499,500,500,500,501,501,501,502,502,502,502,503,503,503,504,504,504,505,505,505,505,506,506,506,507,507,507,508,508,508,508,509,509,509,510,510,510,511,511,511,511,512,512,512,513,513,513,513,514,514,514,515,515,515,516,516,516,516,517,517,517,518,518,518,518,519,519,519,520,520,520,521,521,521,521,522,522,522,523,523,523,523,524,524,524,525,525,525,525,526,526,526,527,527,527,527,528,528,528,529,529,529,529,530,530,530,531,531,531,531,532,532,532,533,533,533,533,534,534,534,535,535,535,535,536,536,536,537,537,537,537,538,538,538,539,539,539,539,540,540,540,540,541,541,541,542,542,542,542,543,543,543,544,544,544,544,545,545,545,545,546,546,546,547,547,547,547,548,548,548,549,549,549,549,550,550,550,550,551,551,551,552,552,552,552,553,553,553,553,554,554,554,555,555,555,555,556,556,556,556,557,557,557,558,558,558,558,559,559,559,559,560,560,560,561,561,561,561,562,562,562,562,563,563,563,563,564,564,564,565,565,565,565,566,566,566,566,567,567,567,568,568,568,568,569,569,569,569,570,570,570,570,571,571,571,571,572,572,572,573,573,573,573,574,574,574,574,575,575,575,575,576,576,576,576,577,577,577,578,578,578,578,579,579,579,579,580,580,580,580,581,581,581,581,582,582,582,582,583,583,583,584,584,584,584,585,585,585,585,586,586,586,586,587,587,587,587,588,588,588,588,589,589,589,589,590,590,590,590,591,591,591,591,592,592,592,593,593,593,593,594,594,594,594,595,595,595,595,596,596,596,596,597,597,597,597,598,598,598,598,599,599,599,599,600,600,600,600,601,601,601,601,602,602,602,602,603,603,603,603,604,604,604,604,605,605,605,605,606,606,606,606,607,607,607,607,608,608,608,608,609,609,609,609,610,610,610,610,611,611,611,611,612,612,612,612,613,613,613,613,614,614,614,614,614,615,615,615,615,616,616,616,616,617,617,617,617,618,618,618,618,619,619,619,619,620,620,620,620,621,621,621,621,622,622,622,622,623,623,623,623,623,624,624,624,624,625,625,625,625,626,626,626,626,627,627,627,627,628,628,628,628,629,629,629,629,629,630,630,630,630,631,631,631,631,632,632,632,632,633,633,633,633,634,634,634,634,634,635,635,635,635,636,636,636,636,637,637,637,637,638,638,638,638,638,639,639,639,639,640,640,640,640,641,641,641,641,642,642,642,642,642,643,643,643,643,644,644,644,644,645,645,645,645,645,646,646,646,646,647,647,647,647,648,648,648,648,648,649,649,649,649,650,650,650,650,651,651,651,651,651,652,652,652,652,653,653,653,653,654,654,654,654,654,655,655,655,655,656,656,656,656,656,657,657,657,657,658,658,658,658,659,659,659,659,659,660,660,660,660,661,661,661,661,661,662,662,662,662,663,663,663,663,664,664,664,664,664,665,665,665,665,666,666,666,666,666,667,667,667,667,668,668,668,668,668,669,669,669,669,670,670,670,670,670,671,671,671,671,672,672,672,672,672,673,673,673,673,674,674,674,674,674,675,675,675,675,676,676,676,676,676,677,677,677,677,677,678,678,678,678,679,679,679,679,679,680,680,680,680,681,681,681,681,681,682,682,682,682,683,683,683,683,683,684,684,684,684,684,685,685,685,685,686,686,686,686,686,687,687,687,687,688,688,688,688,688,689,689,689,689,689,690,690,690,690,691,691,691,691,691,692,692,692,692,692,693,693,693,693,694,694,694,694,694,695,695,695,695,695,696,696,696,696,696,697,697,697,697,698,698,698,698,698,699,699,699,699,699,700,700,700,700,701,701,701,701,701,702,702,702,702,702,703,703,703,703,703,704,704,704,704,705,705,705,705,705,706,706,706,706,706,707,707,707,707,707,708,708,708,708,708,709,709,709,709,710,710,710,710,710,711,711,711,711,711,712,712,712,712,712,713,713,713,713,713,714,714,714,714,714,715,715,715,715,715,716,716,716,716,717,717,717,717,717,718,718,718,718,718,719,719,719,719,719,720,720,720,720,720,721,721,721,721,721,722,722,722,722,722,723,723,723,723,723,724,724,724,724,724,725,725,725,725,725,726,726,726,726,726,727,727,727,727,728,728,728,728,728,729,729,729,729,729,730,730,730,730,730,731,731,731,731,731,732,732,732,732,732,733,733,733,733,733,734,734,734,734,734,735,735,735,735,735,736,736,736,736,736,736,737,737,737,737,737,738,738,738,738,738,739,739,739,739,739,740,740,740,740,740,741,741,741,741,741,742,742,742,742,742,743,743,743,743,743,744,744,744,744,744,745,745,745,745,745,746,746,746,746,746,747,747,747,747,747,748,748,748,748,748,748,749,749,749,749,749,750,750,750,750,750,751,751,751,751,751,752,752,752,752,752,753,753,753,753,753,754,754,754,754,754,754,755,755,755,755,755,756,756,756,756,756,757,757,757,757,757,758,758,758,758,758,758,759,759,759,759,759,760,760,760,760,760,761,761,761,761,761,762,762,762,762,762,762,763,763,763,763,763,764,764,764,764,764,765,765,765,765,765,766,766,766,766,766,766,767,767,767,767,767,768,768,768,768,768,769,769,769,769,769,769,770,770,770,770,770,771,771,771,771,771,772,772,772,772,772,772,773,773,773,773,773,774,774,774,774,774,775,775,775,775,775,775,776,776,776,776,776,777,777,777,777,777,777,778,778,778,778,778,779,779,779,779,779,780,780,780,780,780,780,781,781,781,781,781,782,782,782,782,782,782,783,783,783,783,783,784,784,784,784,784,784,785,785,785,785,785,786,786,786,786,786,786,787,787,787,787,787,788,788,788,788,788,788,789,789,789,789,789,790,790,790,790,790,790,791,791,791,791,791,792,792,792,792,792,792,793,793,793,793,793,794,794,794,794,794,794,795,795,795,795,795,796,796,796,796,796,796,797,797,797,797,797,798,798,798,798,798,798,799,799,799,799,799,799,800,800,800,800,800,801,801,801,801,801,801,802,802,802,802,802,803,803,803,803,803,803,804,804,804,804,804,804,805,805,805,805,805,806,806,806,806,806,806,807,807,807,807,807,807,808,808,808,808,808,809,809,809,809,809,809,810,810,810,810,810,810,811,811,811,811,811,811,812,812,812,812,812,813,813,813,813,813,813,814,814,814,814,814,814,815,815,815,815,815,815,816,816,816,816,816,817,817,817,817,817,817,818,818,818,818,818,818,819,819,819,819,819,819,820,820,820,820,820,821,821,821,821,821,821,822,822,822,822,822,822,823,823,823,823,823,823,824,824,824,824,824,824,825,825,825,825,825,825,826,826,826,826,826,827,827,827,827,827,827,828,828,828,828,828,828,829,829,829,829,829,829,830,830,830,830,830,830,831,831,831,831,831,831,832,832,832,832,832,832,833,833,833,833,833,833,834,834,834,834,834,834,835,835,835,835,835,835,836,836,836,836,836,836,837,837,837,837,837,837,838,838,838,838,838,838,839,839,839,839,839,839,840,840,840,840,840,840,841,841,841,841,841,841,842,842,842,842,842,842,843,843,843,843,843,843,844,844,844,844,844,844,845,845,845,845,845,845,846,846,846,846,846,846,847,847,847,847,847,847,848,848,848,848,848,848,849,849,849,849,849,849,850,850,850,850,850,850,851,851,851,851,851,851,852,852,852,852,852,852,853,853,853,853,853,853,854,854,854,854,854,854,854,855,855,855,855,855,855,856,856,856,856,856,856,857,857,857,857,857,857,858,858,858,858,858,858,859,859,859,859,859,859,860,860,860,860,860,860,860,861,861,861,861,861,861,862,862,862,862,862,862,863,863,863,863,863,863,864,864,864,864,864,864,864,865,865,865,865,865,865,866,866,866,866,866,866,867,867,867,867,867,867,868,868,868,868,868,868,868,869,869,869,869,869,869,870,870,870,870,870,870,871,871,871,871,871,871,871,872,872,872,872,872,872,873,873,873,873,873,873,874,874,874,874,874,874,874,875,875,875,875,875,875,876,876,876,876,876,876,877,877,877,877,877,877,877,878,878,878,878,878,878,879,879,879,879,879,879,879,880,880,880,880,880,880,881,881,881,881,881,881,882,882,882,882,882,882,882,883,883,883,883,883,883,884,884,884,884,884,884,884,885,885,885,885,885,885,886,886,886,886,886,886,886,887,887,887,887,887,887,888,888,888,888,888,888,888,889,889,889,889,889,889,890,890,890,890,890,890,890,891,891,891,891,891,891,892,892,892,892,892,892,892,893,893,893,893,893,893,894,894,894,894,894,894,894,895,895,895,895,895,895,895,896,896,896,896,896,896,897,897,897,897,897,897,897,898,898,898,898,898,898,899,899,899,899,899,899,899,900,900,900,900,900,900,900,901,901,901,901,901,901,902,902,902,902,902,902,902,903,903,903,903,903,903,903,904,904,904,904,904,904,905,905,905,905,905,905,905,906,906,906,906,906,906,906,907,907,907,907,907,907,908,908,908,908,908,908,908,909,909,909,909,909,909,909,910,910,910,910,910,910,910,911,911,911,911,911,911,912,912,912,912,912,912,912,913,913,913,913,913,913,913,914,914,914,914,914,914,914,915,915,915,915,915,915,915,916,916,916,916,916,916,916,917,917,917,917,917,917,918,918,918,918,918,918,918,919,919,919,919,919,919,919,920,920,920,920,920,920,920,921,921,921,921,921,921,921,922,922,922,922,922,922,922,923,923,923,923,923,923,923,924,924,924,924,924,924,924,925,925,925,925,925,925,925,926,926,926,926,926,926,927,927,927,927,927,927,927,928,928,928,928,928,928,928,929,929,929,929,929,929,929,930,930,930,930,930,930,930,931,931,931,931,931,931,931,932,932,932,932,932,932,932,933,933,933,933,933,933,933,934,934,934,934,934,934,934,935,935,935,935,935,935,935,935,936,936,936,936,936,936,936,937,937,937,937,937,937,937,938,938,938,938,938,938,938,939,939,939,939,939,939,939,940,940,940,940,940,940,940,941,941,941,941,941,941,941,942,942,942,942,942,942,942,943,943,943,943,943,943,943,944,944,944,944,944,944,944,944,945,945,945,945,945,945,945,946,946,946,946,946,946,946,947,947,947,947,947,947,947,948,948,948,948,948,948,948,948,949,949,949,949,949,949,949,950,950,950,950,950,950,950,951,951,951,951,951,951,951,952,952,952,952,952,952,952,952,953,953,953,953,953,953,953,954,954,954,954,954,954,954,955,955,955,955,955,955,955,956,956,956,956,956,956,956,956,957,957,957,957,957,957,957,958,958,958,958,958,958,958,958,959,959,959,959,959,959,959,960,960,960,960,960,960,960,961,961,961,961,961,961,961,961,962,962,962,962,962,962,962,963,963,963,963,963,963,963,963,964,964,964,964,964,964,964,965,965,965,965,965,965,965,966,966,966,966,966,966,966,966,967,967,967,967,967,967,967,968,968,968,968,968,968,968,968,969,969,969,969,969,969,969,970,970,970,970,970,970,970,970,971,971,971,971,971,971,971,971,972,972,972,972,972,972,972,973,973,973,973,973,973,973,973,974,974,974,974,974,974,974,975,975,975,975,975,975,975,975,976,976,976,976,976,976,976,976,977,977,977,977,977,977,977,978,978,978,978,978,978,978,978,979,979,979,979,979,979,979,980,980,980,980,980,980,980,980,981,981,981,981,981,981,981,981,982,982,982,982,982,982,982,982,983,983,983,983,983,983,983,984,984,984,984,984,984,984,984,985,985,985,985,985,985,985,985,986,986,986,986,986,986,986,986,987,987,987,987,987,987,987,988,988,988,988,988,988,988,988,989,989,989,989,989,989,989,989,990,990,990,990,990,990,990,990,991,991,991,991,991,991,991,991,992,992,992,992,992,992,992,992,993,993,993,993,993,993,993,993,994,994,994,994,994,994,994,994,995,995,995,995,995,995,995,996,996,996,996,996,996,996,996,997,997,997,997,997,997,997,997,998,998,998,998,998,998,998,998,999,999,999,999,999,999,999,999,1000,1000,1000,1000,1000,1000,1000,1000,1000,1001,1001,1001,1001,1001,1001,1001,1001,1002,1002,1002,1002,1002,1002,1002,1002,1003,1003,1003,1003,1003,1003,1003,1003];
END_VAR

// Globale Variablen/SW_ALZ
{attribute 'qualified_only'}
VAR_GLOBAL
	Bitzer_Scroll_R410a: sw_Einsatzgrenzen := (f_SW_EG_MinVerd := -30, f_SW_EG_MaxVerd := 21, f_SW_EG_MinKond := 25, f_SW_EG_MaxKond := 65, f_SW_EG_BVerd := 12.5, f_SW_EG_BKond := 25, f_SW_EG_CKond := 38, f_SW_EG_DKond := 65, f_SW_EG_EVerd := 21, f_SW_EG_FVerd := 0, f_SW_EG_GKond := 32);
END_VAR

// Globale Variablen/Visu
{attribute 'qualified_only'}
VAR_GLOBAL
	i_Frame_Index:INT;
END_VAR

// Version/Global_Version
{attribute 'TcGenerated'}
// This function has been automatically generated from the project information.
VAR_GLOBAL CONSTANT
	{attribute 'const_non_replaced'}
	{attribute 'linkalways'}
	stLibVersion_GWP_Library : ST_LibVersion := (iMajor := 17, iMinor := 8, iBuild := 1, iRevision := 0, sVersion := '17.8.1');
END_VAR

// Allgemein/Alarm
(*Alarmblock, welcher ein digitaler Ausgang high setzt wenn mind. Ein Alarm anstehend ist und ebenfalls noch die Selbsthaltung der Alarme
*)
FUNCTION_BLOCK Alarm
(*
Versionsverlauf: 
Version		|Autor	|Bemerkung
------------------------------------------------------------------------------------------------------------ 
17.06.00	|Shgb	|erste Freigabe 
17.08.00	|LeaF	|Freigabe

*)
VAR_INPUT
	x_Quittieren:BOOL;//Setzt alle nicht anstehende Alarme auf FALSE
	x_AL1:BOOL;//Alarmeingang 1-16
	x_AL2:BOOL;
	x_AL3:BOOL;
	x_AL4:BOOL;
	x_AL5:BOOL;
	x_AL6:BOOL;
	x_AL7:BOOL;
	x_AL8:BOOL;
	x_AL9:BOOL;
	x_AL10:BOOL;
	x_AL11:BOOL;
	x_AL12:BOOL;
	x_AL13:BOOL;
	x_AL14:BOOL;
	x_AL15:BOOL;
	x_AL16:BOOL;
END_VAR
VAR_OUTPUT	
	x_Aus:BOOL;//Allgemeiner Alarm
	x_AL_1:BOOL;//Alarmausgang 1-16
	x_AL_2:BOOL;
	x_AL_3:BOOL;
	x_AL_4:BOOL;
	x_AL_5:BOOL;
	x_AL_6:BOOL;
	x_AL_7:BOOL;
	x_AL_8:BOOL;
	x_AL_9:BOOL;
	x_AL_10:BOOL;
	x_AL_11:BOOL;
	x_AL_12:BOOL;
	x_AL_13:BOOL;
	x_AL_14:BOOL;
	x_AL_15:BOOL;
	x_AL_16:BOOL;
END_VAR
VAR Persistent
	ax_AL :ARRAY [1..16] OF BOOL;
	ax_Speicher :ARRAY [1..16] OF BOOL;
	i_Arraypos:INT;
	as_Liste: ARRAY [1..16] OF STRING;
END_VAR

//Array füllen
	ax_AL[1]:=x_AL1;
	ax_AL[2]:=x_AL2;
	ax_AL[3]:=x_AL3;
	ax_AL[4]:=x_AL4;
	ax_AL[5]:=x_AL5;
	ax_AL[6]:=x_AL6;
	ax_AL[7]:=x_AL7;
	ax_AL[8]:=x_AL8;
	ax_AL[9]:=x_AL9;
	ax_AL[10]:=x_AL10;
	ax_AL[11]:=x_AL11;
	ax_AL[12]:=x_AL12;
	ax_AL[13]:=x_AL13;
	ax_AL[14]:=x_AL14;
	ax_AL[15]:=x_AL15;
	ax_AL[16]:=x_AL16;
	
	
	
	
	
	
	
//Quittieren
	IF x_Quittieren THEN
		FOR i_Arraypos:=1 TO 16 DO
			ax_Speicher[i_Arraypos]:=FALSE;
		END_FOR
	END_IF

//Alarme Setzen
	FOR i_Arraypos:=1 TO 16 DO
		IF ax_AL[i_Arraypos] THEN
			ax_Speicher[i_Arraypos]:=TRUE;
		END_IF
	END_FOR

//Ausgäne setzen
	x_AL_1:=ax_Speicher[1];
	x_AL_2:=ax_Speicher[2];
	x_AL_3:=ax_Speicher[3];
	x_AL_4:=ax_Speicher[4];
	x_AL_5:=ax_Speicher[5];
	x_AL_6:=ax_Speicher[6];
	x_AL_7:=ax_Speicher[7];
	x_AL_8:=ax_Speicher[8];
	x_AL_9:=ax_Speicher[9];
	x_AL_10:=ax_Speicher[10];
	x_AL_11:=ax_Speicher[11];
	x_AL_12:=ax_Speicher[12];
	x_AL_13:=ax_Speicher[13];
	x_AL_14:=ax_Speicher[14];
	x_AL_15:=ax_Speicher[15];
	x_AL_16:=ax_Speicher[16];
	
	x_Aus:=x_al_1 OR 
			x_al_2 OR 
			x_al_3 OR 
			x_al_4 OR
			x_al_5 OR
			x_al_6 OR
			x_al_7 OR
			x_al_8 OR
			x_al_9 OR
			x_al_10 OR
			x_al_11 OR
			x_al_12 OR
			x_al_13 OR
			x_al_14 OR
			x_al_15 OR
			x_AL_16;

END_FUNCTION_BLOCK

// Allgemein/COUNT
(*Je nachdem wieviele digitale Eingänge true sind, wird er analoge Ausgang hochgezählt. Ist kein Eingang auf true, bleibt der Ausgang auf 0.
Der Counter ist auf max. 8 digitale Eingänge ausgelegt.
*)
FUNCTION_BLOCK COUNT
(*
Versionsverlauf: 
Version		|Autor	|Bemerkung
------------------------------------------------------------------------------------------------------------ 
17.05.00	|KuzR	|erste Freigabe  
17.08.00	|LeaF	|Freigabe

*)
VAR_INPUT	
	x_Ein_1:BOOL;//8 Digitale Eingänge
	x_Ein_2:BOOL;
	x_Ein_3:BOOL;
	x_Ein_4:BOOL;
	x_Ein_5:BOOL;
	x_Ein_6:BOOL;
	x_Ein_7:BOOL;
	x_Ein_8:BOOL;
END_VAR
VAR_OUTPUT
	i_Aus:Int;//Ausganng in Int
END_VAR
VAR	
END_VAR

	i_Aus:=0;
// Ausgang zählt hoch, wenn Eingang true ist
	IF x_Ein_1 THEN
		i_Aus:=i_Aus+1;
	END_IF
	
	IF x_Ein_2 THEN
		i_Aus:=i_Aus+1;
	END_IF
	
	IF x_Ein_3 THEN
		i_Aus:=i_Aus+1;
	END_IF
	
	IF x_Ein_4 THEN
		i_Aus:=i_Aus+1;
	END_IF
	
	IF x_Ein_5 THEN
		i_Aus:=i_Aus+1;
	END_IF
	
	IF x_Ein_6 THEN
		i_Aus:=i_Aus+1;
	END_IF
	
	IF x_Ein_7 THEN
		i_Aus:=i_Aus+1;
	END_IF
	
	IF x_Ein_8 THEN
		i_Aus:=i_Aus+1;
	END_IF

END_FUNCTION_BLOCK

// Allgemein/MUX_B
(*Anhand von 4 digitalen Eingängen wird entschieden, welcher von 4 analogen Werten (Real) auf den analogen Ausgang (Real) geschrieben wird.
Der kleinere Eingang hat immer Priorität für das Schreiben des Ausganges. Wenn keine Eingänge auf true sind, dann Augang auf 0.

*)
FUNCTION_BLOCK MUX_B
(*
Versionsverlauf: 
Version		|Autor	|Bemerkung
------------------------------------------------------------------------------------------------------------ 
17.06.00	|KuzR	|erste Freigabe  
17.08.00	|LeaF	|Freigabe

*)
VAR_INPUT
	f_Ein_1:REAL;//Eingangswerte 1-4 in Real
	f_Ein_2:REAL;
	f_Ein_3:REAL;
	f_Ein_4:REAL;
	x_Ein_1:BOOL;//Digitaler Eingang 1
	x_Ein_2:BOOL;//Digitaler Eingang 2
	x_Ein_3:BOOL;//Digitaler Eingang 3
	x_Ein_4:BOOL;//Digitaler Eingang 4
END_VAR
VAR_OUTPUT
	f_Aus:REAL;//Ausgang in Real
END_VAR
VAR
END_VAR

	f_Aus:=0;
//Wenn 1.Eingang True, dann Wert1
	IF x_Ein_1  THEN
		f_Aus := f_Ein_1;		
//Ansonsen wird beim Ausgang Wert zwei geschrieben
	ELSIF x_Ein_2 THEN
		f_Aus := f_Ein_2;		
	ELSIF x_Ein_3 THEN
		f_Aus := f_Ein_3;		
	ELSIF x_Ein_4 THEN
		f_Aus := f_Ein_4;							
	END_IF

END_FUNCTION_BLOCK

// Allgemein/MUX_D_INT
(*Anhand von 3 analogen Eingangswerten (Integer)wird mit dem i_Sel entschieden, welcher von den 3 Eingängen auf den analogen Ausgang (Integer) geschrieben wird.
*)
FUNCTION_BLOCK MUX_D_INT
(*
Versionsverlauf: 
Version		|Autor	|Bemerkung
------------------------------------------------------------------------------------------------------------ 
17.05.00	|KuzR	|erste Freigabe  
17.08.00	|LeaF	|Freigabe

*)
VAR_INPUT
	i_Ein_1:INT;//Eingangswert 1 als Int
	i_Ein_2:INT;//Eingangswert 2 als Int
	i_Ein_3:INT; //Eingangswert 3 als Int
	i_Sel:INT;// Auswahl Selector
	
END_VAR
VAR_OUTPUT
	i_Aus:INT;//Ausgang als Int
END_VAR
VAR
END_VAR

//Mit Select Auswählen, welcher Eingang auf Ausgang geschrieben wird
	CASE i_sel OF
		1: i_Aus:= i_Ein_1;
		2: i_Aus:= i_Ein_2;
		3: i_Aus:= i_Ein_3;
	ELSE	
//Wenn Select <3 oder >0, dann Ausgang 0
		i_Aus:=0;
	END_CASE

END_FUNCTION_BLOCK

// Allgemein/MUX_D_REAL
(*Anhand von 3 analogen Eingangswerten (Real)wird mit dem i_Sel entschieden, welcher von den 3 Eingängen auf den analogen Ausgang (Real) geschrieben wird.
*)
FUNCTION_BLOCK MUX_D_REAL
(*
Versionsverlauf: 
Version		|Autor	|Bemerkung
------------------------------------------------------------------------------------------------------------ 
17.06.00	|ShgB	|erste Freigabe  
17.08.00	|LeaF	|Freigabe

*)
VAR_INPUT
	f_Ein_1:REAL;//Eingangswert 1 als Real
	f_Ein_2:REAL;//Eingangswert 2 als Real
	f_Ein_3:REAL;//Eingangswert 3 als Real
	i_Sel:INT;// Auswahl Selector
	
END_VAR
VAR_OUTPUT
	f_Aus:REAL;//Ausgang in Real
END_VAR
VAR
END_VAR

//Mit Select Auswählen, welcher Eingang auf Ausgang geschrieben wird
	CASE i_sel OF
		1: f_Aus:= f_Ein_1;
		2: f_Aus:= f_Ein_2;
		3: f_Aus:= f_Ein_3;
	ELSE
		
//Wenn Select <0 oder >3, dann Ausgang 0
		f_Aus:=0;
	END_CASE

END_FUNCTION_BLOCK

// Allgemein/NULL
(*Wenn der analoge Eingang (Real) genau 0 ist, wird der digitale Ausgang auf true gesetzt, ansonsten auf false.
*)
FUNCTION_BLOCK NULL
(*
Versionsverlauf: 
Version		|Autor	|Bemerkung
------------------------------------------------------------------------------------------------------------ 
17.06.00	|KuzR	|erste Freigabe  
17.08.00	|LeaF	|Freigabe

*)
VAR_INPUT
	i_Ein:REAL;//Eingangswert in Real
END_VAR
VAR_OUTPUT
	x_Aus:BOOL;//Digitaler Ausgang
END_VAR
VAR
END_VAR

//Wenn 0 gleich Ausgang true, ansonsten false
	x_Aus:=i_Ein =0;

END_FUNCTION_BLOCK

// Allgemein/SWITCH_INT
(*Ist der digitale Eingang auf false, wird der erste analoge Eingangswert (Int) in den analogen Ausgang (Int) geschrieben. 
Ist der digitale Eingang auf true, wird der zweite analoge Eingangswert (Int) in den analogen Ausgang (Int) geschrieben.
*)
FUNCTION_BLOCK SWITCH_INT
(*
Versionsverlauf: 
Version		|Autor	|Bemerkung
------------------------------------------------------------------------------------------------------------ 
17.05.00	|KuzR	|erste Freigabe  
17.08.00	|LeaF	|Freigabe

*)
VAR_INPUT
	x_Ein:BOOL;//Digitaler Eingang
	i_Ein_1:INT;//Analoger Eingangswert 1 als Int
	i_Ein_2:INT;//Analoger Eingangswert 2 als Int
END_VAR
VAR_OUTPUT
	i_Aus:INT;//Analoger Ausgangswert als Int
END_VAR
VAR	
END_VAR

	IF x_Ein THEN		
//Wenn Eingang True, Wert_2 in Ausgang
		i_Aus:= i_Ein_2;	
	ELSE	
//Wenn Eingang false, Wert_1 in Ausgang
		i_Aus:= i_Ein_1;
	END_IF

END_FUNCTION_BLOCK

// Allgemein/SWITCH_REAL
(*Ist der digitale Eingang auf false, wird der erste analoge Eingangswert (Real) in den analogen Ausgang (Real) geschrieben. 
Ist der digitale Eingang auf true, wird der zweite analoge Eingangswert (Real) in den analogen Ausgang (Real) geschrieben.
*)
FUNCTION_BLOCK SWITCH_REAL
(*
Versionsverlauf: 
Version		|Autor	|Bemerkung
------------------------------------------------------------------------------------------------------------ 
17.05.00	|KuzR	|erste Freigabe  
17.08.00	|LeaF	|Freigabe

*)
VAR_INPUT
	x_Ein:BOOL;//Digitaler Eingang
	f_Ein_1:REAL;//Analoger Eingangswert 1 als Real
	f_Ein_2	:REAL;//Analoger Eingangswert 2 als Real
END_VAR
VAR_OUTPUT
	f_Aus:REAL;//Analoger Ausgangswert als Real
END_VAR
VAR	
END_VAR

	IF x_Ein THEN		
//Wenn Eingang True, Wert_2 in Ausgang
		f_Aus:= f_Ein_2;	
	ELSE	
//Wenn Eingang false, Wert_1 in Ausgang
		f_Aus:= f_Ein_1;
	END_IF

END_FUNCTION_BLOCK

// Allgemein/Toggle
(*Mit einer positiven Flanke auf den x_Toggle Eingang wird der Wert des Ausgangs x_Aus zwischen FALSE und TRUE gwechselt.
Mit dem x_Reset Eingang kann der Ausgang auf FALSE geschrieben werden. 
*)
FUNCTION_BLOCK Toggle
(*
Versionsverlauf: 
Version		|Autor	|Bemerkung
------------------------------------------------------------------------------------------------------------ 
17.06.00	|Shgb	|erste Freigabe  
17.08.00	|LeaF	|Freigabe

*)
VAR_INPUT
	x_Toggle:BOOL;//Wechselt den Wert des Ausgangs bei einer positiven Flanke
	x_Reset:BOOL;//Setzt den Ausgang auf FALSE
END_VAR
VAR_OUTPUT
	x_Aus:BOOL;//Ausgang
END_VAR
VAR PERSISTENT
	x_Speicher: BOOL;
END_VAR
VAR
	x_Flanke:BOOL;
END_VAR

//Toggle mit Flankenerkennung
	IF x_Toggle AND NOT x_Flanke THEN
		x_Speicher:= NOT x_Speicher;
	END_IF
	x_Flanke:=x_Toggle;

//Reset
	IF x_Reset THEN
		x_Speicher:=FALSE;
	END_IF
	
//Ausgang schreiben
	x_Aus:=x_Speicher;

END_FUNCTION_BLOCK

// Converters/Converter2Punkt
(*Der Eingang f_Ein wird anhand des Bereiches von f_Ein_Min f_Ein_Max auf den Bereich f_Aus_Min und f_Aus_Max berechnet und auf den Ausgang f_Aus gegeben.
*)
FUNCTION_BLOCK Converter2Punkt
(*
Versionsverlauf: 
Version		|Autor	|Bemerkung
------------------------------------------------------------------------------------------------------------ 
17.06.00	|ShgB	|erste Freigabe 
17.06.01	|ShgB	|von Integer auf Real geändert 
17.08.00	|LeaF	|Freigabe	

*)
VAR_INPUT
	f_Ein:REAL;//Eingang
	f_Ein_Min:REAL;//Eingangsbereich Minimum
	f_Ein_Max:REAL;//Eingangsbereich Maximum
	f_Aus_Min:REAL;//Ausgangsbereich Minimum
	f_Aus_Max:REAL;//Ausgangsbereich Maximum
END_VAR
VAR_OUTPUT
	f_Aus:REAL;//Ausgang
END_VAR
VAR
END_VAR

IF f_Ein_Max-f_Ein_Min <> 0 THEN
	f_Aus:=(f_Aus_Max-f_Aus_Min)/(f_Ein_Max-f_Ein_Min)*(f_Ein-f_Ein_Min)+f_Aus_Min;
ELSE
	f_Aus:=f_Aus_Max;
END_IF

END_FUNCTION_BLOCK

// Math/Maximum
(*Gibt den grössten der angeschlossenen Werten aus.
*)
FUNCTION_BLOCK Maximum
(*
Versionsverlauf: 
Version		|Autor	|Bemerkung
------------------------------------------------------------------------------------------------------------ 
17.06.00	|Shgb	|erste Freigabe 
17.06.01	|ShgB	|von Integer auf Real geändert	 
17.08.00	|LeaF	|Freigabe

*)
VAR_INPUT
	f_Ein1 :REAL:=0.00001;//Wert 1
	f_Ein2 :REAL:=0.00001;//Wert 2
	f_Ein3 :REAL:=0.00001;//Wert 3
	f_Ein4 :REAL:=0.00001;//Wert 4
	f_Ein5 :REAL:=0.00001;//Wert 5
	f_Ein6 :REAL:=0.00001;//Wert 6
	f_Ein7 :REAL:=0.00001;//Wert 7
	f_Ein8 :REAL:=0.00001;//Wert 8
END_VAR
VAR_OUTPUT
	f_Aus:REAL;//Grösste Wert
END_VAR
VAR
	i_Arraypos:INT;
	af_Array: ARRAY [1..8] OF REAL;
END_VAR

// Werte in Array platzieren
	af_Array[1]:=f_Ein1;
	af_Array[2]:=f_Ein2;
	af_Array[3]:=f_Ein3;
	af_Array[4]:=f_Ein4;
	af_Array[5]:=f_Ein5;
	af_Array[6]:=f_Ein6;
	af_Array[7]:=f_Ein7;
	af_Array[8]:=f_Ein8;
	
//Zahlen die kleiner als 0 sind
	f_Aus := af_Array[1];	
	
//Auswertung der grössten Zahl
	FOR i_Arraypos:=2 TO 8 DO
		IF af_Array[i_Arraypos] >= f_Aus AND af_Array[i_Arraypos] <> 0.00001 THEN
			f_Aus := af_Array[i_Arraypos];
		END_IF
	END_FOR

END_FUNCTION_BLOCK

// Converters/Int_to_Druck
(*Der analoge Wert der Eingangskarte wird von einem 16 bit Integer in einen REAL Wert umgewandelt und ein Offset dazu addiert.
Standardmässig ist der Eingangsbereich von 0 - 32767 eingestellt. Sollte dieser nicht übereinstimmen kann der Bereich angepasst werden.
*)
FUNCTION_BLOCK Int_to_Druck
(*
Versionsverlauf: 
Version		|Autor	|Bemerkung
------------------------------------------------------------------------------------------------------------ 
17.06.00	|Shgb	|erste Freigabe  
17.08.00	|LeaF	|Freigabe

*)
VAR_INPUT
	i_Ein:INT;//Digitaler Eingangswert
END_VAR
VAR_INPUT PERSISTENT
	i_Ein_Min:INT:=0;//Eingangsbereich Minimum
	i_Ein_Max:INT:=32767;//Eingangsbereich Maximum
	f_Aus_Min:REAL;//Minimum des Drucktransmitters
	f_Aus_Max:REAL;//Maximum des Drucktransmitters
	f_Offset:REAL;//Offset der dazu addiert wird
END_VAR
VAR_OUTPUT
	f_Aus:REAL;//Druck im REAL Format
END_VAR
VAR
END_VAR

IF i_Ein_Max-i_Ein_Min <> 0 THEN
	f_Aus:=(f_Aus_Max-f_Aus_Min)/(i_Ein_Max-i_Ein_Min)*(i_Ein-i_Ein_Min)+f_Aus_Min+f_Offset;
ELSE
	f_Aus:=f_Aus_Min;
END_IF

END_FUNCTION_BLOCK

// Converters/Int_to_Temperature
(*Wandelt die Temperatur im INT Format, die von der Eingangskarte kommt, in eine Temperatur in REAL Format um und rechnet einen Offset dazu.
*)
FUNCTION_BLOCK Int_to_Temperature
(*
Versionsverlauf: 
Version		|Autor	|Bemerkung
------------------------------------------------------------------------------------------------------------ 
17.06.00	|Shgb	|erste Freigabe  
17.08.00	|LeaF	|Freigabe

*)
VAR_INPUT
	i_Ein:INT;//Temperatur von Karte
END_VAR
VAR_INPUT PERSISTENT
	f_Offset:REAL;//Offset der dazu addiert wird
END_VAR
VAR_OUTPUT
	f_Temperatur:REAL;//Ausgang REAL
END_VAR
VAR
END_VAR

f_Temperatur:=i_Ein/10.0+f_Offset;

END_FUNCTION_BLOCK

// Converters/Prozent_to_Int
(*Wandelt eine Prozentangabe vom Format REAL in eine Integer Zahl für die analoge Augangskarte um.
Standardmässig ist der Eingangsbereich von 0 - 32767 eingestellt. Sollte dieser nicht übereinstimmen kann der Bereich angepasst werden.
*)
FUNCTION_BLOCK Prozent_to_Int
(*
Versionsverlauf: 
Version		|Autor	|Bemerkung
------------------------------------------------------------------------------------------------------------ 
17.06.00	|Shgb	|erste Freigabe 
17.08.00	|LeaF	|Freigabe 

*)
VAR_INPUT
	f_Ein:REAL;//Eingang in Prozent
END_VAR
VAR_INPUT PERSISTENT
	i_Aus_Min:INT:=0;//Eingangsbereich Minimum
	i_Aus_Max:INT:=32767;//eingangsbereich Maximum
END_VAR
VAR_OUTPUT
	f_Aus:INT;//Ausgang
END_VAR
VAR
END_VAR

f_Aus:=real_to_int((i_Aus_Max-i_Aus_Min)*f_Ein/100.0);

END_FUNCTION_BLOCK

// Converters/Time_to_Timestruct
(*Wandelt die Eingangsvariable vom Typ TIME in ein TIMESTRUCT um.
*)
FUNCTION_BLOCK Time_to_Timestruct
(*
Versionsverlauf: 
Version		|Autor	|Bemerkung
------------------------------------------------------------------------------------------------------------ 
17.06.00	|Shgb	|erste Freigabe 	 
17.08.00	|LeaF	|Freigabe

*)
VAR_INPUT
	t_Ein:TIME;//Eingang
END_VAR
VAR_OUTPUT
	t_Aus:timestruct;//Ausgang
END_VAR
VAR
	OT:OTSTRUCT;
END_VAR

OT:=TIME_TO_OTSTRUCT(t_Ein);
t_Aus.wMilliseconds:=ot.wMilliseconds;
t_Aus.wSecond:=ot.wSecond;
t_Aus.wMinute:=ot.wMinute;
t_Aus.wHour:=ot.wHour;
t_Aus.wDay:=ot.wDay+ot.wWeek*7;

END_FUNCTION_BLOCK

// Converters/Timestruct_to_Time
(*Wandelt einen TIMESTRUCT in die Ausgangsvariable vom Typ TIME um.
*)
FUNCTION_BLOCK Timestruct_to_Time
(*
Versionsverlauf: 
Version		|Autor	|Bemerkung
------------------------------------------------------------------------------------------------------------ 
17.06.00	|Shgb	|erste Freigabe  
17.08.00	|LeaF	|Freigabe	

*)
VAR_INPUT
	t_Ein:timestruct;//Eingang
END_VAR
VAR_OUTPUT
	t_Aus:TIME;//Ausgang
END_VAR
VAR
END_VAR

t_Aus:=DINT_TO_TIME(t_Ein.wMilliseconds
					+ t_Ein.wSecond*1000
					+ t_Ein.wMinute*1000*60
					+ t_Ein.wHour*1000*60*60
					+ t_Ein.wDay*1000*60*60*24);

END_FUNCTION_BLOCK

// Druck_Temp/R1234ze
(*Wandelt den Druck in die Entsprechende Temperatur um. Die Druck-Temperatur Werte sind in der Nassdampftabelle in den Globalen Variablen hinterlegt.
*)
FUNCTION_BLOCK R1234ze
(*
Versionsverlauf: 
Version		|Autor	|Bemerkung
------------------------------------------------------------------------------------------------------------ 
17.06.00	|Shgb	|erste Freigabe 
17.06.01	|ShgB	|von Integer auf Real geändert	 
17.08.00	|LeaF	|Freigabe

*)
VAR_INPUT
	f_ND:REAL;//Druck für Verdampfungstemperatur
	f_HD:REAL;//Druck für Kondensationstemperatur
END_VAR
VAR_OUTPUT
	f_VerdTemp:REAL;//Verdampfungstemperatur
	f_KondTemp:REAL;//Kondensationstemperatur
END_VAR
VAR
END_VAR

//Niederdruck
	f_VerdTemp:=Nassdampftabelle.R1234ze[REAL_TO_INT(f_ND*100)+100]/10.0;
	
//Hochdruck
	f_KondTemp:=Nassdampftabelle.R1234ze[REAL_TO_INT(f_HD*100)+100]/10.0;

END_FUNCTION_BLOCK

// Druck_Temp/R134a
(*Wandelt den Druck in die Entsprechende Temperatur um. Die Druck-Temperatur Werte sind in der Nassdampftabelle in den Globalen Variablen hinterlegt.
*)
FUNCTION_BLOCK R134a
(*
Versionsverlauf: 
Version		|Autor	|Bemerkung
------------------------------------------------------------------------------------------------------------ 
17.06.00	|Shgb	|erste Freigabe 
17.06.01	|ShgB	|von Integer auf Real geändert	 
17.08.00	|LeaF	|Freigabe

*)
VAR_INPUT
	f_ND:REAL;//Druck für Verdampfungstemperatur
	f_HD:REAL;//Druck für Kondensationstemperatur
END_VAR
VAR_OUTPUT
	f_VerdTemp:REAL;//Verdampfungstemperatur
	f_KondTemp:REAL;//Kondensationstemperatur
END_VAR
VAR
END_VAR

//Niederdruck
	f_VerdTemp:=Nassdampftabelle.R134a[REAL_TO_INT(f_ND*100)+100]/10.0;
	
//Hochdruck
	f_KondTemp:=Nassdampftabelle.R134a[REAL_TO_INT(f_HD*100)+100]/10.0;

END_FUNCTION_BLOCK

// Druck_Temp/R410a
(*Wandelt den Druck in die Entsprechende Temperatur um. Die Druck-Temperatur Werte sind in der Nassdampftabelle in den Globalen Variablen hinterlegt.
*)
FUNCTION_BLOCK R410a
(*
Versionsverlauf: 
Version		|Autor	|Bemerkung
------------------------------------------------------------------------------------------------------------ 
17.06.00	|Shgb	|erste Freigabe 
17.06.01	|ShgB	|von Integer auf Real geändert	 
17.08.00	|LeaF	|Freigabe

*)
VAR_INPUT
	f_ND:REAL;//Druck für Verdampfungstemperatur
	f_HD:REAL;//Druck für Kondensationstemperatur
END_VAR
VAR_OUTPUT
	f_VerdTemp:REAL;//Verdampfungstemperatur
	f_KondTemp:REAL;//Kondensationstemperatur
END_VAR
VAR
END_VAR

//Niederdruck
	f_VerdTemp:=Nassdampftabelle.R410a[REAL_TO_INT(f_ND*100)+100]/10.0;
	
//Hochdruck
	f_KondTemp:=Nassdampftabelle.R410a[REAL_TO_INT(f_HD*100)+100]/10.0;

END_FUNCTION_BLOCK

// Handschaltungen/HS_Bool
(*Handschaltung für BOOL. 0=> Aus, 1=> Ein und 2=> Automatik.
*)
FUNCTION_BLOCK HS_Bool
(*
Versionsverlauf: 
Version		|Autor	|Bemerkung
------------------------------------------------------------------------------------------------------------ 
17.06.00	|Shgb	|erste Freigabe   
17.08.00	|LeaF	|Freigabe

*)
VAR_INPUT
	x_Ein:BOOL;//Eingang
END_VAR
VAR_INPUT PERSISTENT
	i_Modus:INT;//Modusvorgabe
END_VAR
VAR_OUTPUT
	x_Aus:BOOL;//Ausgang
END_VAR
VAR
END_VAR
VAR CONSTANT
	Ein:INT:=1;
	Aus:INT:=0;
	Auto:INT:=2;
END_VAR

CASE i_Modus OF
	Ein:
		x_Aus:=TRUE;
	Aus:
		x_Aus:=FALSE;
	Auto:
		x_Aus:=x_Ein;
ELSE
	x_Aus:=FALSE;
END_CASE;

END_FUNCTION_BLOCK

// Handschaltungen/HS_Int
(*Handschaltung für INT. 1=> Manuell und 2=> Automatik.
*)
FUNCTION_BLOCK HS_Int
(*
Versionsverlauf: 
Version		|Autor	|Bemerkung
------------------------------------------------------------------------------------------------------------ 
17.06.00	|Shgb	|erste Freigabe   
17.08.00	|LeaF	|Freigabe

*)
VAR_INPUT
	i_Ein:INT;//Eingang
END_VAR
VAR_INPUT PERSISTENT
	i_Manu:INT;//Manuelle Sollstellung
	i_Modus:INT;//Modusvorgabe
END_VAR
VAR_OUTPUT
	i_Aus:INT;//Ausgang
END_VAR
VAR
END_VAR
VAR CONSTANT
	Ein:INT:=1;
	Aus:INT:=0;
	Auto:INT:=2;
END_VAR

CASE i_Modus OF
	Ein:
		i_Aus:=i_Manu;
	Auto:
		i_Aus:=i_Ein;
ELSE
	i_Aus:=0;
END_CASE;

END_FUNCTION_BLOCK

// Handschaltungen/HS_Real
(*Handschaltung für REAL. 1=> Manuell und 2=> Automatik.
*)
FUNCTION_BLOCK HS_Real
(*
Versionsverlauf: 
Version		|Autor	|Bemerkung
------------------------------------------------------------------------------------------------------------ 
17.06.00	|Shgb	|erste Freigabe   
17.08.00	|LeaF	|Freigabe

*)
VAR_INPUT
	f_Ein:REAL;//Eingang
END_VAR
VAR_INPUT PERSISTENT
	f_Manu:REAL;//Manuelle Sollstellung
	i_Modus:INT;//Modusvorgabe
END_VAR
VAR_OUTPUT
	f_Aus:real;//Ausgang
END_VAR
VAR
END_VAR
VAR CONSTANT
	Ein:INT:=1;
	Aus:INT:=0;
	Auto:INT:=2;
END_VAR

CASE i_Modus OF
	Ein:
		f_Aus:=f_Manu;
	Auto:
		f_Aus:=f_Ein;
ELSE
	f_Aus:=0;
END_CASE;

END_FUNCTION_BLOCK

// Heizen_Kuehlen/FG_Heizen
(* Mit der Tagesschaltuhr wird der Tag_Nacht Sollwert bestimmt. Schaltuhr Ein = Nachtbetrieb. Der Funktionsblock wird mit dem Eingang x_Akt aktiviert.
 Unterschreitet die Aussentemperatur und die gemittelte AT den einstellbaren Sollwert
 in der fix eingestellten Zeit von 5 Minuten, schaltet der Einschaltbefehl bis die beiden Temperatur Werte
 der eingestellten Sollwert wieder überschreiten. 
 *)
FUNCTION_BLOCK FG_Heizen
(*
Versionsverlauf: 
Version		|Autor	|Bemerkung
------------------------------------------------------------------------------------------------------------ 
17.07.00	|KuzR	|erste Freigabe  
17.08.00	|LeaF	|Freigabe

*)
VAR_INPUT 
	x_Nacht:BOOL;//Ein=Nacht, Aus=Tag
	f_AT:REAL;//Aussentemperatur
	f_RT_AT:REAL;//Berechnete Aussentemperatur
END_VAR
VAR_INPUT PERSISTENT
	x_Akt_FB:BOOL := TRUE;//Aktivierung FB
	f_SW_Tag:REAL := 20;//Sollwert Tag
	f_SW_Nacht:REAL := 16;//Sollwert Nacht
END_VAR
VAR_OUTPUT
	x_EB:BOOL;//Einschaltbefehl
END_VAR
VAR
	f_Aus_SW_Tag_Nacht:REAL;
	x_EIN_Timer:BOOL;
	Timer:TON;
	MUX_B: MUX_B;
	CLK_D: CLK_D;
	Timestruct_to_Time: Timestruct_to_Time;
	t_time: TIME;
	x_FG_Tag:BOOL;
	x_FG_Nacht:BOOL;
END_VAR

//Nachtakivierung
	x_FG_Nacht:=x_Akt_FB AND x_Nacht;
	
//Tagaktivierung	
	x_FG_Tag:=x_Akt_FB AND NOT x_Nacht;
	
//Tag/Nacht Umschaltung
	MUX_B(
	f_Ein_1:=f_SW_Tag , 
	f_Ein_2:=f_SW_Nacht , 
	x_Ein_1:=x_FG_Tag , 
	x_Ein_2:=x_FG_Nacht , 
	f_Aus=>f_Aus_SW_Tag_Nacht );	

//Temperaturen Abfrage Tag_Nacht und Timer einschalten
	x_EIN_Timer:= x_Akt_FB AND  f_AT < f_Aus_SW_Tag_Nacht AND f_RT_AT < f_Aus_SW_Tag_Nacht;
		
//Timer Restzeit für Abfrage AT und SW
	Timer(in:=x_EIN_Timer , pt:=T#5M);	

//Einschaltbefehl 	
	x_EB:=Timer.Q;

END_FUNCTION_BLOCK

// Uhren/CLK_D
(*Uhr mit Tagesprogramm. Einschaltzeit => t_Ein.wHour, t_ein.wMinute und Ausschaltzeit => t_Aus.wHour und t_Aus.wMinute. Eingabe im Timestruct Format.
Vergleicht Ein- und Ausschaltzeit mit der Globalen_Uhr(Globale Variable)
*)
FUNCTION_BLOCK CLK_D
(*
Versionsverlauf: 
Version		|Autor	|Bemerkung
------------------------------------------------------------------------------------------------------------ 
17.06.00	|KuzR	|erste Freigabe 
17.08.00	|LeaF	|Freigabe

*)
VAR_INPUT Persistent
	t_Ein:timestruct;//Eingabe Einschaltzeit 
	t_Aus:timestruct;//Eingabe Ausschaltzeit 
END_VAR
VAR_OUTPUT
	x_Aus:BOOL;//Digitaler Ausgang		 
END_VAR
VAR
END_VAR

//schaltet jeden Tag ein, eingestell e Zeit  
	IF Globale_Uhr.systemtimestruct.wHour = t_Ein.wHour AND
 	   Globale_Uhr.systemtimestruct.wMinute >= t_Ein.wMinute THEN
			x_Aus:= TRUE;
	END_IF
				
//schaltet jeden Tag wieder aus, eingestellte Zeit			
	IF 	Globale_Uhr.systemtimestruct.wHour = t_Aus.wHour AND
		Globale_Uhr.systemtimestruct.wMinute >= t_Aus.wMinute THEN
			x_Aus:= FALSE;
	END_IF

END_FUNCTION_BLOCK

// Heizen_Kuehlen/FG_Kuehlen
(* Mit der Tagesschaltuhr wird der Tag_Nacht Sollwert bestimmt. Schaltuhr Ein = Nachtbetrieb. Der Funktionsblock wird mit dem Eingang x_Akt aktiviert.
 Überschreitet die Aussentemperatur und die gemittelte AT den einstellbaren Sollwert
 in der fix eingestellten Zeit von 5 Min und der Eingang x_Absch_Hz_Kue war länger nicht angezogen, schaltet der Einschaltbefehl bis die beiden Temperatur Werte
 der eingestellten Sollwert wieder unterschreiten. 
 *)
FUNCTION_BLOCK FG_Kuehlen
(*
Versionsverlauf: 
Version		|Autor	|Bemerkung
------------------------------------------------------------------------------------------------------------ 
17.07.00	|KuzR	|erste Freigabe  
17.08.00	|LeaF	|Freigabe

*)
VAR_INPUT 
	f_AT:REAL;//Aussentemperatur
	f_RT_AT:REAL;//Berechnete Aussentemperatur
END_VAR
VAR_INPUT PERSISTENT
	x_Akt_FB:BOOL := true;//Aktivierung FB
	x_Nacht: BOOL;//Ein=Nacht, Aus=Tag
	f_SW_Tag:REAL := 10;//Sollwert Tag
	f_SW_Nacht:REAL := 10;//Sollwert Nacht
	x_Absch_HZ_Kue:BOOL;//Abschaltung HZ und Kühlen
END_VAR
VAR_OUTPUT
	x_EB:BOOL;//Einschaltbefehl
END_VAR
VAR
	f_Aus_SW_Tag_Nacht:REAL;
	x_Tag_Nacht:BOOL;
	x_EIN_Timer:BOOL;
	Timer:TON;
	MUX_B: MUX_B;
	CLK_D: CLK_D;
	Timestruct_to_Time: Timestruct_to_Time;
	t_time: TIME;
	x_FG_Tag:BOOL;//Freigabe Tag
	x_FG_Nacht:BOOL;//Freigabe Nacht
END_VAR

//Nachtakivierung
	x_FG_Nacht:=x_Akt_FB AND x_Nacht;
	
//Tagaktivierung	
	x_FG_Tag:=x_Akt_FB AND NOT x_Nacht;
	
//Tag/Nacht Umschaltung
	MUX_B(
	f_Ein_1:=f_SW_Tag , 
	f_Ein_2:=f_SW_Nacht , 
	x_Ein_1:=x_FG_Tag , 
	x_Ein_2:=x_FG_Nacht , 
	f_Aus=>f_Aus_SW_Tag_Nacht );	

//Temperaturen Abfrage Tag_Nacht und Timer einschalten
	x_EIN_Timer:= x_Akt_FB AND  f_AT > f_Aus_SW_Tag_Nacht AND f_RT_AT > f_Aus_SW_Tag_Nacht AND NOT x_Absch_HZ_Kue;
		
//Timer Restzeit für Abfrage AT und SW
	Timer(in:=x_EIN_Timer , pt:=T#5M);	

//Einschaltbefehl 	
	x_EB:=Timer.Q;

END_FUNCTION_BLOCK

// Heizen_Kuehlen/GR_2
//Kühlkurve, mit 2 AT-Punkten wird ein Tag, bzw. Nachtsollwert berechnet. Referenpunkt T01 muss grösser sein Als T02
//Umschaltbar Tag/Nacht Aktivierung. Sollwert Max und Min Begrenzung. 
FUNCTION_BLOCK GR_2
(*
Versionsverlauf: 
Version		|Autor	|Bemerkung
------------------------------------------------------------------------------------------------------------ 
17.06.00	|KuzR	|erste Freigabe  
17.08.00	|LeaF	|Freigabe

*)
VAR_INPUT
	f_AT:REAL;//Aussentempertur
	x_Akt_Nacht:BOOL;//Nachtakivierung	
END_VAR
VAR_INPUT PERSISTENT
	f_RefPunkt_TO1:REAL;//Referenzpunkt T01 AT
	f_SW_W1_Tag:REAL;//Sollwertpunkt 1 Tag
	f_SW_W1_Nacht:REAL;//Sollwertpunkt 1 Nacht
	f_RefPunkt_TO2:REAL;//Referenzpunkt T02 AT
	f_SW_W2_Tag:REAL;//Sollwertpunkt 2 Tag
	f_SW_W2_Nacht:REAL;//Sollwertpunkt 1 Nacht
	f_SW_Max:REAL;//Sollwert Max.
	f_SW_Min:REAL;//Sollwert Min.
END_VAR
VAR_OUTPUT
	f_SW_Ber:REAL;//Ausgang Sollwert
END_VAR
	
VAR
	
	Converter2Punkt: Converter2Punkt;
END_VAR

//T01 muss Höher sein als T02
//Aussentemperatur T2-T1, Tag
//Aussentemperatur < T1 oder Aussentemperatur > T2 für Min/Max Begrenzung
	IF NOT x_Akt_Nacht AND  f_RefPunkt_TO2 <= f_AT AND f_RefPunkt_TO1 > f_AT OR NOT x_Akt_Nacht AND f_AT < f_RefPunkt_TO1 OR NOT x_Akt_Nacht AND f_AT > f_RefPunkt_TO2  THEN 
		Converter2Punkt(
	f_Ein:=f_AT , 
	f_Ein_Min:=f_RefPunkt_TO1 , 
	f_Ein_Max:=f_RefPunkt_TO2 , 
	f_Aus_Min:=f_SW_W1_Tag , 
	f_Aus_Max:=f_SW_W2_Tag , 
	f_Aus=>f_SW_Ber );
	END_IF
	
//Aussentemperatur T2-T1, Nacht
//Aussentemperatur < T1 oder Aussentemperatur > T2 für Min/Max Begrenzung
	IF  x_Akt_Nacht AND  
		f_RefPunkt_TO2 <= f_AT AND 
		f_RefPunkt_TO1 > f_AT OR  x_Akt_Nacht AND f_AT < f_RefPunkt_TO1 OR x_Akt_Nacht AND f_AT < f_RefPunkt_TO1 OR  x_Akt_Nacht AND f_AT > f_RefPunkt_TO2  THEN 
		Converter2Punkt(
	f_Ein:=f_AT , 
	f_Ein_Min:=f_RefPunkt_TO1 , 
	f_Ein_Max:=f_RefPunkt_TO2 , 
	f_Aus_Min:=f_SW_W1_Nacht , 
	f_Aus_Max:=f_SW_W2_Nacht , 
	f_Aus=>f_SW_Ber );
	END_IF
	
//Min/Max Begrenzung 
	f_SW_Ber := LIMIT(f_SW_Min,f_SW_Ber, f_SW_Max);

END_FUNCTION_BLOCK

// Heizen_Kuehlen/GR_4_mit_RE
(* Heizkurve mit Raumeinfluss vergleicht Aussentemperatur zwischen den Sollwerten. Referenzpunkt T01 muss die kleinste Temperatur-,bzw. T04 die grösste Temperatur sein.
 Anhand von vier AT Punkten wird der Tag-, bzw. Nachtsollwert berechnet.
 Umschaltbar Tag/Nacht Aktivierung. Sollwert mit  Max und Min Begrenzung. Maximale negative Korrektur (i_MaxKorrNeg) muss zwingend als negativen Wert eingegeben werden und Maximale positive  Korrektur als positiven Wert.
*)
FUNCTION_BLOCK GR_4_mit_RE
(*
Versionsverlauf: 
Version		|Autor	|Bemerkung
------------------------------------------------------------------------------------------------------------ 
17.06.00	|KuzR	|erste Freigabe  
17.08.00	|LeaF	|Freigabe

*)
VAR_INPUT
	f_AT:REAL; //Aussentemperatur
	x_Akt_Nacht:BOOL;	// Nachtakivierung
	f_MT_Raum:REAL; // Raumtemperatur
END_VAR
VAR_INPUT PERSISTENT	
	f_RefPunkt_TO1:REAL; // Referenzpunkt T01 AT
	f_SW_W1_Tag:REAL; // Sollwertpunkt 1 Tag
	f_SW_W1_Nacht:REAL; // Sollwertpunkt 1 Nacht
	f_RefPunkt_TO2:REAL; // Referenzpunkt T02 AT
	f_SW_W2_Tag:REAL; // Sollwertpunkt 2 Tag
	f_SW_W2_Nacht:REAL; // Sollwertpunkt 2 Nacht
	f_RefPunkt_TO3:REAL; // Referenzpunkt T03 AT
	f_SW_W3_Tag:REAL; // Sollwertpunkt 3 Tag
	f_SW_W3_Nacht:REAL; // Sollwertpunkt 3 Nacht
	f_RefPunkt_TO4:REAL; // Referenzpunkt T04 AT
	f_SW_W4_Tag:REAL; // Sollwertpunkt 4 Tag
	f_SW_W4_Nacht:REAL; // Sollwertpunkt 4 Nacht
	f_SW_Max:REAL; // Sollwert Max.
	f_SW_Min:REAL; //Sollwert Min.
	f_KorrFaktor:REAL;  // Korrekturfaktor
	i_MaxKorrPos:INT; // Max. Pos. Korrektur(muss positiver Wert sein)
	i_MaxKorrNeg:INT; // Max. Neg. Korrektur(muss negativer Wert sein)
	f_SW_Raum:REAL;	// Sollwert Raum
END_VAR
VAR_OUTPUT
	f_SW_Ber:REAL; // Sollwert Berechnung
	f_SW_Korr:REAL; // Korrigierte Sollwertberechnung
END_VAR
VAR
	f_Diff:REAL;
	f_Diff_faktor:REAL;
	Converter2Punkt: Converter2Punkt;
END_VAR

//Aussentemperatur T4-T3, Tag
//Aussentemperatur > T4, für Max Sollwert Berechnung
	IF NOT x_Akt_Nacht AND f_RefPunkt_TO4 > f_AT AND f_RefPunkt_TO3 <= f_AT OR NOT x_Akt_Nacht AND f_AT >= f_RefPunkt_TO4 THEN
		Converter2Punkt( 
	f_Ein:=f_AT , 
	f_Ein_Min:=f_RefPunkt_TO3 , 
	f_Ein_Max:=f_RefPunkt_TO4 , 
	f_Aus_Min:=f_SW_W3_Tag , 
	f_Aus_Max:=f_SW_W4_Tag , 
	f_Aus=>f_SW_Ber );
	END_IF
//Aussentemperatur T4-T3, Nacht
//Aussentemperatur > T4, für Max Sollwert Berechnung
	IF x_Akt_Nacht AND f_RefPunkt_TO4 > f_AT AND f_RefPunkt_TO3 <= f_AT OR x_Akt_Nacht AND f_AT >= f_RefPunkt_TO4 THEN
		Converter2Punkt(
	f_Ein:=f_AT , 
	f_Ein_Min:=f_RefPunkt_TO3 , 
	f_Ein_Max:=f_RefPunkt_TO4 , 
	f_Aus_Min:=f_SW_W3_Nacht , 
	f_Aus_Max:=f_SW_W4_Nacht , 
	f_Aus=>f_SW_Ber );
	END_IF
//Aussentemperatur T3-T2, Tag
	IF NOT x_Akt_Nacht AND  f_RefPunkt_TO3 > f_AT AND f_RefPunkt_TO2 <= f_AT THEN
		Converter2Punkt(
	f_Ein:=f_AT , 
	f_Ein_Min:=f_RefPunkt_TO2 , 
	f_Ein_Max:=f_RefPunkt_TO3 , 
	f_Aus_Min:=f_SW_W2_Tag , 
	f_Aus_Max:=f_SW_W3_Tag , 
	f_Aus=>f_SW_Ber );
	END_IF
//Aussentemperatur T3-T2, Nacht
	IF x_Akt_Nacht AND  f_RefPunkt_TO3 > f_AT AND f_RefPunkt_TO2 <= f_AT THEN
		Converter2Punkt(
	f_Ein:=f_AT , 
	f_Ein_Min:=f_RefPunkt_TO2 , 
	f_Ein_Max:=f_RefPunkt_TO3 , 
	f_Aus_Min:=f_SW_W2_Nacht , 
	f_Aus_Max:=f_SW_W3_Nacht , 
	f_Aus=>f_SW_Ber );
	END_IF	
//Aussentemperatur T2-T1, Tag
//Aussentemperatur < T1, für Min Sollwert Berechnung
	IF NOT x_Akt_Nacht AND f_RefPunkt_TO2 > f_AT AND f_RefPunkt_TO1 <= f_AT OR NOT x_Akt_Nacht AND f_AT < f_RefPunkt_TO1  THEN
		Converter2Punkt(
	f_Ein:=f_AT , 
	f_Ein_Min:=f_RefPunkt_TO1 , 
	f_Ein_Max:=f_RefPunkt_TO2 , 
	f_Aus_Min:=f_SW_W1_Tag , 
	f_Aus_Max:=f_SW_W2_Tag , 
	f_Aus=>f_SW_Ber );
	END_IF
//Aussentemperatur T2-T1, Nacht
//Aussentemperatur < T1, für Min Sollwert Berechnung
	IF x_Akt_Nacht AND f_RefPunkt_TO2 > f_AT AND f_RefPunkt_TO1 <= f_AT OR x_Akt_Nacht AND f_AT < f_RefPunkt_TO1  THEN
		Converter2Punkt(
	f_Ein:=f_AT , 
	f_Ein_Min:=f_RefPunkt_TO1 , 
	f_Ein_Max:=f_RefPunkt_TO2 , 
	f_Aus_Min:=f_SW_W1_Nacht , 
	f_Aus_Max:=f_SW_W2_Nacht , 
	f_Aus=>f_SW_Ber );
	END_IF

//Korrektur Raumtemperatur
	f_Diff:= f_SW_Raum-f_MT_Raum;
	
//Maximale_Minimale Korrektur
	IF f_Diff > i_MaxKorrPos THEN
		f_Diff:=i_MaxKorrPos;
	END_IF
	IF f_Diff < i_MaxKorrNeg THEN
		f_Diff:=i_MaxKorrNeg;
	END_IF
	
	f_Diff_faktor:=f_Diff*f_KorrFaktor;
	
//Begrenzung für positive und negative Begerenzung
	IF f_Diff_faktor > i_MaxKorrPos THEN
		f_Diff_faktor:=i_MaxKorrPos;
	END_IF
	IF f_Diff_faktor < i_MaxKorrNeg THEN
		f_Diff_faktor:=i_MaxKorrNeg;
	END_IF
	
//Korrrigierter Sollwert	
	f_SW_Korr:=f_SW_Ber + f_Diff_faktor ;

//Max Begrenzung 	
	IF f_SW_Korr >= f_SW_Max THEN
		f_SW_Korr:=f_SW_Max; 
	END_IF	
//Min Begrenzung 
	IF f_SW_Korr < f_SW_Min THEN
		f_SW_Korr:=f_SW_Min;
	END_IF

END_FUNCTION_BLOCK

// Heizen_Kuehlen/GR_4_ohne_RE
(* Heizkurve ohne Raumeinfluss vergleicht Aussentemperatur zwischen den Sollwerten. Referenzpunkt T01 muss die kleinste Temperatur-,bzw. T04 die grösste Temperatur sein.
 Anhand von vier AT Punkten wird der Tag-, bzw. Nachtsollwert berechnet.
 Umschaltbar Tag/Nacht Aktivierung. Sollwert MAX und MIN Begrenzung.
*)
FUNCTION_BLOCK GR_4_ohne_RE
(*
Versionsverlauf: 
Version		|Autor	|Bemerkung
------------------------------------------------------------------------------------------------------------ 
17.06.00	|KuzR	|erste Freigabe  
17.08.00	|LeaF	|Freigabe

*)
VAR_INPUT
	f_AT:REAL; //Aussentemperatur
	x_Akt_Nacht:BOOL;//Nachtakivierung
END_VAR
VAR_INPUT PERSISTENT
	f_RefPunkt_TO1:REAL;//Referenzpunkt T01 AT
	f_SW_W1_Tag:REAL;//Sollwertpunkt 1 Tag
	f_SW_W1_Nacht:REAL;//Sollwertpunkt 1 Nacht
	f_RefPunkt_TO2:REAL;//Referenzpunkt T02 AT
	f_SW_W2_Tag:REAL;//Sollwertpunkt 2 Tag
	f_SW_W2_Nacht:REAL;//Sollwertpunkt 2 Nacht
	f_RefPunkt_TO3:REAL;//Referenzpunkt T03 AT
	f_SW_W3_Tag:REAL;//Sollwertpunkt 3 Tag
	f_SW_W3_Nacht:REAL;//Sollwertpunkt 3 Nacht
	f_RefPunkt_TO4:REAL;//Referenzpunkt T04 AT
	f_SW_W4_Tag:REAL;//Sollwertpunkt 4 Tag
	f_SW_W4_Nacht:REAL;//Sollwertpunkt 4 Nacht
	f_SW_Max:REAL;//Sollwert Max.
	f_SW_Min:REAL;//Sollwert Min.
END_VAR
VAR_OUTPUT
	f_SW_Ber:REAL;//Sollwert Berechnung
END_VAR
VAR
	Converter2Punkt: Converter2Punkt;
END_VAR

//Aussentemperatur T4-T3, Tag
//Aussentemperatur > T4, für Max Sollwert Berechnung
	IF NOT x_Akt_Nacht AND f_RefPunkt_TO4 > f_AT AND f_RefPunkt_TO3 <= f_AT OR NOT x_Akt_Nacht AND f_AT >= f_RefPunkt_TO4 THEN
		Converter2Punkt( 
	f_Ein:=f_AT , 
	f_Ein_Min:=f_RefPunkt_TO3 , 
	f_Ein_Max:=f_RefPunkt_TO4 , 
	f_Aus_Min:=f_SW_W3_Tag , 
	f_Aus_Max:=f_SW_W4_Tag , 
	f_Aus=>f_SW_Ber );
	END_IF
//Aussentemperatur T4-T3, Nacht
//Aussentemperatur > T4, für Max Sollwert Berechnung
	IF x_Akt_Nacht AND f_RefPunkt_TO4 > f_AT AND f_RefPunkt_TO3 <= f_AT OR x_Akt_Nacht AND f_AT >= f_RefPunkt_TO4 THEN
		Converter2Punkt(
	f_Ein:=f_AT , 
	f_Ein_Min:=f_RefPunkt_TO3 , 
	f_Ein_Max:=f_RefPunkt_TO4 , 
	f_Aus_Min:=f_SW_W3_Nacht , 
	f_Aus_Max:=f_SW_W4_Nacht , 
	f_Aus=>f_SW_Ber );
	END_IF
//Aussentemperatur T3-T2, Tag
	IF NOT x_Akt_Nacht AND  f_RefPunkt_TO3 > f_AT AND f_RefPunkt_TO2 <= f_AT THEN
		Converter2Punkt(
	f_Ein:=f_AT , 
	f_Ein_Min:=f_RefPunkt_TO2 , 
	f_Ein_Max:=f_RefPunkt_TO3 , 
	f_Aus_Min:=f_SW_W2_Tag , 
	f_Aus_Max:=f_SW_W3_Tag , 
	f_Aus=>f_SW_Ber );
	END_IF
//Aussentemperatur T3-T2, Nacht
	IF x_Akt_Nacht AND  f_RefPunkt_TO3 > f_AT AND f_RefPunkt_TO2 <= f_AT THEN
		Converter2Punkt(
	f_Ein:=f_AT , 
	f_Ein_Min:=f_RefPunkt_TO2 , 
	f_Ein_Max:=f_RefPunkt_TO3 , 
	f_Aus_Min:=f_SW_W2_Nacht , 
	f_Aus_Max:=f_SW_W3_Nacht , 
	f_Aus=>f_SW_Ber );
	END_IF	
//Aussentemperatur T2-T1, Tag
//Aussentemperatur < T1, für Min Sollwert Berechnung
	IF NOT x_Akt_Nacht AND f_RefPunkt_TO2 > f_AT AND f_RefPunkt_TO1 <= f_AT OR NOT x_Akt_Nacht AND f_AT < f_RefPunkt_TO1  THEN
		Converter2Punkt(
	f_Ein:=f_AT , 
	f_Ein_Min:=f_RefPunkt_TO1 , 
	f_Ein_Max:=f_RefPunkt_TO2 , 
	f_Aus_Min:=f_SW_W1_Tag , 
	f_Aus_Max:=f_SW_W2_Tag , 
	f_Aus=>f_SW_Ber );
	END_IF
//Aussentemperatur T2-T1, Nacht
//Aussentemperatur < T1, für Min Sollwert Berechnung
	IF x_Akt_Nacht AND f_RefPunkt_TO2 > f_AT AND f_RefPunkt_TO1 <= f_AT OR x_Akt_Nacht AND f_AT < f_RefPunkt_TO1  THEN
		Converter2Punkt(
	f_Ein:=f_AT , 
	f_Ein_Min:=f_RefPunkt_TO1 , 
	f_Ein_Max:=f_RefPunkt_TO2 , 
	f_Aus_Min:=f_SW_W1_Nacht , 
	f_Aus_Max:=f_SW_W2_Nacht , 
	f_Aus=>f_SW_Ber );
	END_IF

//Min/Max Begrenzung 	
	f_SW_Ber := LIMIT(f_SW_Min,f_SW_Ber, f_SW_Max);

END_FUNCTION_BLOCK

// Heizen_Kuehlen/REG2_HEIZEN
(*2 Punkt Regler Heizen
Für Direkt, x_Akt auf true, schaltet der Ausgang auf true. Ist der eingegebene Sollwert addiert mit dem Einschaltpunkt(zB -2) grösser oder gleich der Messtemperatur,
schaltet der digitale Ausgang auf true. Ist der Sollwert addiert mit dem Ausschaltpunkt kleiner oder gleich dem Messwert, schaltet der digitale Ausganf auf false.
*)
FUNCTION_BLOCK REG2_HEIZEN
(*
Versionsverlauf: 
Version		|Autor	|Bemerkung
------------------------------------------------------------------------------------------------------------ 
17.06.00	|KuzR	|erste Freigabe  
17.08.00	|LeaF	|Freigabe

*)
VAR_INPUT
	f_MT:REAL;//Eingang Messwert
END_VAR
VAR_INPUT PERSISTENT
	f_SW:REAL;//Eingang Sollwert
	f_Einschaltpunkt:REAL;//Eingang Einschaltpunkt
	f_Ausschaltpunkt:REAL;//Eingang Ausschaltpunkt
	x_Akt:BOOL;//Direkt-Indirekt Aktivierung
END_VAR
VAR_OUTPUT
	x_Aus:BOOL;//Digitaler Ausgang
END_VAR
VAR
END_VAR

//Direkt- Indirekt Schaltung
	IF   NOT x_Akt THEN 
		x_Aus:=FALSE;
//Einschalten
	ELSIF  f_MT <= f_SW + f_Einschaltpunkt THEN
		x_Aus:= TRUE;
//Ausschalten	
	ELSIF	f_MT  >= f_SW + f_Ausschaltpunkt THEN
		x_Aus:= FALSE;
	END_IF

END_FUNCTION_BLOCK

// Heizen_Kuehlen/REG2_KUEHLEN
(*2 Punkt Regler Kühlen
Für Direkt, x_Akt auf true, schaltet der Ausgang auf true. Ist der eingegebene Sollwert addiert mit dem Einschaltpunkt(zB -2) kleiner oder gleich der Messtemperatur,
schaltet der digitale Ausgang auf true. Ist der Sollwert addiert mit dem Ausschaltpunkt grösser oder gleich dem Messwert, schaltet der digitale Ausganf auf false.
*)
FUNCTION_BLOCK REG2_KUEHLEN
(*
Versionsverlauf: 
Version		|Autor	|Bemerkung
------------------------------------------------------------------------------------------------------------ 
17.06.00	|KuzR	|erste Freigabe  
17.08.00	|LeaF	|Freigabe

*)
VAR_INPUT
	f_MT:REAL;//Eingang Messwert
END_VAR
VAR_INPUT PERSISTENT
	f_SW:REAL;//Eingang Sollwert
	f_Einschaltpunkt:REAL;//Eingang Einschaltpunkt
	f_Ausschaltpunkt:REAL;//Eingang Ausschaltpunkt
	x_Akt:BOOL;//Direkt-Indirekt Aktivierung
END_VAR
VAR_OUTPUT
	x_Aus:BOOL;//Digitaler Ausgang
END_VAR
VAR
END_VAR

//Direkt- Indirekt Schaltung
	IF   NOT x_Akt THEN 
		x_Aus:=FALSE;	
//Einschalten
	ELSIF  f_MT >= f_SW + f_Einschaltpunkt THEN
		x_Aus:= TRUE;	
//Ausschalten	
	ELSIF	f_MT  <= f_SW + f_Ausschaltpunkt THEN
		x_Aus:= FALSE;	
	END_IF

END_FUNCTION_BLOCK

// Heizen_Kuehlen/RT_AT_48
(*Berechnet die gemittelte Aussentemperatur. Die Datensätze für die Mittelwertberechnung ist auf 48 Datensätze ausgelegt.
x_start für die Initialisierung der Aussentemperatur. Mit t_time kann die Zeit bestimmt werden, wann einen Wert ins Array geschrieben werden kann.
*)
FUNCTION_BLOCK RT_AT_48
(*
Versionsverlauf: 
Version		|Autor	|Bemerkung
------------------------------------------------------------------------------------------------------------ 
17.07.00	|KuzR	|erste Freigabe  
17.08.00	|LeaF	|Freigabe

*)
VAR_INPUT
	x_start: BOOL;//Start für die  Initialisierung
	f_AT:REAL;//Eingang Aussentemperatur
END_VAR
VAR_INPUT PERSISTENT	
	t_time:timestruct;//Zeiteingabe 1h oder 24h
END_VAR
VAR_OUTPUT
	f_AT_RT: REAL;//Ausgang gemittelt
END_VAR
VAR 
	i_Ind: INT;
	f_Summe:REAL;
	timer:ton;
	daten:ARRAY [1..i_Datensaetze] OF REAL;
	Timestruct_to_Time:Timestruct_to_Time;	
	x_Flanke: BOOL;
END_VAR
VAR CONSTANT
	i_Datensaetze:INT:=48;
END_VAR

//Für Aussentemperatur Initialisierung muss x_start gedrückt werden
	 IF x_start  THEN
//Grösse des Array für den Mittelwert bestimmen
		 FOR i_Ind:= 1 TO I_DATENSAETZE DO
			 daten[i_Ind]:= f_AT;
		 END_FOR
	 END_IF
	x_start:=FALSE;
//Timestruct to Time
	timestruct_to_time(t_Ein:=t_time);
//Timer läuft immer
	Timer(IN := NOT Timer.Q, PT :=timestruct_to_time.t_Aus/48 );

	IF Timer.Q THEN
    f_Summe := 0;
//die neuen Temperaturwerte werden ins Array geschrieben
    FOR i_Ind := I_DATENSAETZE TO 2 BY -1  DO
        Daten[i_Ind] := Daten[i_Ind - 1];
        f_Summe := f_Summe + Daten[i_Ind];
    END_FOR
//Rechentemperatur berechnen
    Daten[1] := f_AT;
    f_Summe := f_Summe + f_AT;
    f_AT_RT:=f_summe / I_DATENSAETZE;
	END_IF

END_FUNCTION_BLOCK

// Initialisierung/Globale_Zeit
FUNCTION_BLOCK Globale_Zeit
(*
Versionsverlauf: 
Version		|Autor	|Bemerkung
------------------------------------------------------------------------------------------------------------ 
17.06.00	|KuzR	|erste Freigabe 
17.06.01	|ShgB	|Date and Time ergänzt 
17.08.00	|LeaF	|Freigabe

*)
VAR_INPUT Persistent
	tzi_ZeitZone:ST_TimeZoneInformation :=WEST_EUROPE_TZI;
END_VAR
VAR_OUTPUT		 
END_VAR
VAR
	  fbgetSystemTime:getsystemtime;
  	  fileTime:T_FILETIME;
	  
      eTzID:E_TimeZoneID := eTimeZoneID_Unknown;
      fbToLocal:FB_FileTimeToTzSpecificLocalTime;
	  tzInfo:ST_TimeZoneInformation;
END_VAR

//CPU Zeit
	fbgetSystemTime	(timeLoDW=>fileTime.dwLowDateTime, timeHiDW=>fileTime.dwHighDateTime );
	
//Zeitumrechnung
	fbToLocal( in := filetime , tzInfo := tzi_ZeitZone );
	
//Globale Variable, Aktuelle Uhrzeit
	Globale_Uhr.systemtimestruct := FILETIME_TO_systemtime( fbToLocal.out  );
	Globale_Uhr.systemDateAndTime:= FILETIME_TO_DT(fbToLocal.out);

END_FUNCTION_BLOCK

// Math/Average
(*Gibt den Durchschnitt der angeschlossenen Werten aus.
*)
FUNCTION_BLOCK Average
(*
Versionsverlauf: 
Version		|Autor	|Bemerkung
------------------------------------------------------------------------------------------------------------ 
17.06.00	|Shgb	|erste Freigabe  
17.08.00	|LeaF	|Freigabe

*)
VAR_INPUT
	f_Ein1 :REAL:=0.00001;//Wert 1
	f_Ein2 :REAL:=0.00001;//Wert 2
	f_Ein3 :REAL:=0.00001;//Wert 3
	f_Ein4 :REAL:=0.00001;//Wert 4
	f_Ein5 :REAL:=0.00001;//Wert 5
	f_Ein6 :REAL:=0.00001;//Wert 6
	f_Ein7 :REAL:=0.00001;//Wert 7
	f_Ein8 :REAL:=0.00001;//Wert 8
END_VAR
VAR_OUTPUT
	f_Aus:REAL;//Durchschnitt
END_VAR
VAR
	i_Arraypos:INT;
	af_Array: ARRAY [1..8] OF REAL;
	COUNT: COUNT;
END_VAR

// Werte in Array platzieren
	af_Array[1]:=f_Ein1;
	af_Array[2]:=f_Ein2;
	af_Array[3]:=f_Ein3;
	af_Array[4]:=f_Ein4;
	af_Array[5]:=f_Ein5;
	af_Array[6]:=f_Ein6;
	af_Array[7]:=f_Ein7;
	af_Array[8]:=f_Ein8;
	
//Zurücksetzen
	f_Aus:=0;
	
//Anzahl Eingänge zählen
	COUNT(
	x_Ein_1:= f_Ein1<>0.00001, //0.00001 bedeutet nicht aktiv
	x_Ein_2:= f_Ein2<>0.00001, 
	x_Ein_3:= f_Ein3<>0.00001, 
	x_Ein_4:= f_Ein4<>0.00001, 
	x_Ein_5:= f_Ein5<>0.00001, 
	x_Ein_6:= f_Ein6<>0.00001, 
	x_Ein_7:= f_Ein7<>0.00001, 
	x_Ein_8:= f_Ein8<>0.00001);
	
//Summe bilden
	FOR i_Arraypos:=1 TO count.i_Aus DO
		f_Aus:=f_Aus+af_Array[i_Arraypos];
	END_FOR
	
//Durchschnitt berechnen
	IF count.i_Aus >0 THEN
		f_Aus:=f_Aus/count.i_Aus;
	END_IF

END_FUNCTION_BLOCK

// Math/Filter
(*Berechnet die gefilterte Aussentemperatur. x_start für die Initialisierung der Aussentemperatur. Mit t_time kann die Zeit bestimmt werden, wann einen Wert ins Array geschrieben werden kann.
*)
FUNCTION_BLOCK Filter
(*
Versionsverlauf:
Version		|Autor	|Bemerkung
------------------------------------------------------------------------------------------------------------ 
17.07.00	|KuzR	|erste Freigabe  
17.08.00	|LeaF	|Freigabe

*)
VAR_INPUT
	x_start: BOOL;//Start für die  Initialisierung
	f_AT:REAL;//Eingang Aussentemperatur
END_VAR
VAR_INPUT PERSISTENT	
	t_time:timestruct := (wHour := 1);//Takt, wenn ein AT Wert geschrieben wird
END_VAR
VAR_OUTPUT
	f_Aus: REAL;//Ausgang gefiltert
END_VAR
VAR 
	i_Ind: INT;
	f_Summe:REAL;
	timer:ton;
	daten:ARRAY [1..i_Datensaetze] OF REAL;
	Timestruct_to_Time:Timestruct_to_Time;	
	x_Flanke: BOOL;
END_VAR
VAR CONSTANT
	i_Datensaetze:INT:=48;
END_VAR

//Für Aussentemperatur Initialisierung muss x_start gedrückt werden
	 IF x_start  THEN
//Grösse des Array für den Mittelwert bestimmen
		 FOR i_Ind:= 1 TO I_DATENSAETZE DO
			 daten[i_Ind]:= f_AT;
		 END_FOR
	 END_IF
		x_start:=FALSE;
//Timestruct to Time
	timestruct_to_time(t_Ein:=t_time);
//Timer läuft immer
	Timer(IN := NOT Timer.Q, PT :=timestruct_to_time.t_Aus );

	IF Timer.Q THEN
    f_Summe := 0;
//die neuen Temperaturwerte werden ins Array geschrieben
    FOR i_Ind := I_DATENSAETZE TO 2 BY -1  DO
        Daten[i_Ind] := Daten[i_Ind - 1];
        f_Summe := f_Summe + Daten[i_Ind];
    END_FOR
//Rechentemperatur berechnen
    Daten[1] := f_AT;
    f_Summe := f_Summe + f_AT;
    f_Aus:=f_summe / I_DATENSAETZE;
	END_IF

END_FUNCTION_BLOCK

